LIN {X 0,Y 313.862,Z 653.442,A -85,B 0,C 180,E1 -16164.593,E2 -16164.593} C_VEL
LIN {X 0,Y 312.967,Z 666.014,A -85,B 0,C 180,E1 -16165.653,E2 -16165.653} C_VEL
LIN {X 0,Y 311.886,Z 679.603,A -85,B 0,C 180,E1 -16167.108,E2 -16167.108} C_VEL
LIN {X 0,Y 310.731,Z 691.302,A -85,B 0,C 180,E1 -16168.655,E2 -16168.655} C_VEL
LIN {X 0,Y 309.643,Z 702.145,A -85,B 0,C 180,E1 -16170.419,E2 -16170.419} C_VEL
LIN {X 0,Y 308.883,Z 708.95,A -85,B 0,C 180,E1 -16171.72,E2 -16171.72} C_VEL
LIN {X 0,Y 307.8,Z 712.897,A -85,B 0,C 180,E1 -16172.513,E2 -16172.513} C_VEL
LIN {X 0,Y 304.339,Z 719.014,A -85,B 0,C 180,E1 -16173.825,E2 -16173.825} C_VEL
LIN {X 0,Y 300.937,Z 724.622,A -85,B 0,C 180,E1 -16175.238,E2 -16175.238} C_VEL
LIN {X 0,Y 299.968,Z 727.754,A -85,B 0,C 180,E1 -16176.177,E2 -16176.177} C_VEL
LIN {X 0,Y 299.269,Z 734.632,A -85,B 0,C 180,E1 -16178.655,E2 -16178.655} C_VEL
LIN {X 0,Y 298.891,Z 739.258,A -85,B 0,C 180,E1 -16180.781,E2 -16180.781} C_VEL
LIN {X 0,Y 298.646,Z 742.834,A -85,B 0,C 180,E1 -16182.893,E2 -16182.893} C_VEL
LIN {X 0,Y 298.627,Z 745.46,A -85,B 0,C 180,E1 -16184.997,E2 -16184.997} C_VEL
LIN {X 0,Y 298.833,Z 747.584,A -85,B 0,C 180,E1 -16187.781,E2 -16187.781} C_VEL
LIN {X 0,Y 299.31,Z 748.208,A -85,B 0,C 180,E1 -16190.54,E2 -16190.54} C_VEL
LIN {X 0,Y 300.074,Z 747.31,A -85,B 0,C 180,E1 -16193.276,E2 -16193.276} C_VEL
LIN {X 0,Y 301.251,Z 744.941,A -85,B 0,C 180,E1 -16195.987,E2 -16195.987} C_VEL
LIN {X 0,Y 302.374,Z 742.07,A -85,B 0,C 180,E1 -16198.047,E2 -16198.047} C_VEL
LIN {X 0,Y 304.129,Z 737.027,A -85,B 0,C 180,E1 -16200.663,E2 -16200.663} C_VEL
LIN {X 0,Y 305.674,Z 732.008,A -85,B 0,C 180,E1 -16202.636,E2 -16202.636} C_VEL
LIN {X 0,Y 307.809,Z 724.674,A -85,B 0,C 180,E1 -16204.912,E2 -16204.912} C_VEL
LIN {X 0,Y 309.873,Z 716.852,A -85,B 0,C 180,E1 -16206.839,E2 -16206.839} C_VEL
LIN {X 0,Y 312.038,Z 707.448,A -85,B 0,C 180,E1 -16208.745,E2 -16208.745} C_VEL
LIN {X 0,Y 314.263,Z 696.794,A -85,B 0,C 180,E1 -16210.486,E2 -16210.486} C_VEL
LIN {X 0,Y 316.318,Z 685.009,A -85,B 0,C 180,E1 -16212.023,E2 -16212.023} C_VEL
LIN {X 0,Y 318.24,Z 671.492,A -85,B 0,C 180,E1 -16213.408,E2 -16213.408} C_VEL
LIN {X 0,Y 319.562,Z 658.715,A -85,B 0,C 180,E1 -16214.439,E2 -16214.439} C_VEL
LIN {X 0,Y 320.44,Z 645.691,A -85,B 0,C 180,E1 -16215.235,E2 -16215.235} C_VEL
LIN {X 0,Y 320.888,Z 631.299,A -85,B 0,C 180,E1 -16215.863,E2 -16215.863} C_VEL
LIN {X 0,Y 322.128,Z 601.129,A -85,B 0,C 180,E1 -16216.863,E2 -16216.863} C_VEL
LIN {X 0,Y 317.545,Z 592.238,A -85,B 0,C 180,E1 -16218.074,E2 -16218.074} C_VEL
LIN {X 0,Y 311.17,Z 581.718,A -85,B 0,C 180,E1 -16219.887,E2 -16219.887} C_VEL
LIN {X 0,Y 308.467,Z 577.764,A -85,B 0,C 180,E1 -16220.724,E2 -16220.724} C_VEL
LIN {X 0,Y 306.134,Z 574.422,A -85,B 0,C 180,E1 -16221.491,E2 -16221.491} C_VEL
LIN {X 0,Y 305.23,Z 573.248,A -85,B 0,C 180,E1 -16221.792,E2 -16221.792} C_VEL
LIN {X 0,Y 302.984,Z 570.401,A -85,B 0,C 180,E1 -16222.579,E2 -16222.579} C_VEL
LIN {X 0,Y 302.035,Z 568.615,A -85,B 0,C 180,E1 -16222.97,E2 -16222.97} C_VEL
LIN {X 0,Y 299.778,Z 566.635,A -85,B 0,C 180,E1 -16223.784,E2 -16223.784} C_VEL
LIN {X 0,Y 298.652,Z 564.26,A -85,B 0,C 180,E1 -16224.329,E2 -16224.329} C_VEL
LIN {X 0,Y 298.46,Z 563.308,A -85,B 0,C 180,E1 -16224.494,E2 -16224.494} C_VEL
LIN {X 0,Y 298.467,Z 563.298,A -85,B 0,C 180,E1 -16228.096,E2 -16228.096} C_VEL
LIN {X 0,Y 298.393,Z 563.303,A -85,B 0,C 180,E1 -16232.018,E2 -16232.018} C_VEL
LIN {X 0,Y 298.417,Z 563.307,A -85,B 0,C 180,E1 -16236.071,E2 -16236.071} C_VEL
LIN {X 0,Y 298.407,Z 563.307,A -85,B 0,C 180,E1 -16239.487,E2 -16239.487} C_VEL
LIN {X 0,Y 298.397,Z 563.316,A -85,B 0,C 180,E1 -16243.104,E2 -16243.104} C_VEL
LIN {X 0,Y 298.402,Z 563.315,A -85,B 0,C 180,E1 -16246.922,E2 -16246.922} C_VEL
LIN {X 0,Y 298.492,Z 563.489,A -85,B 0,C 180,E1 -16249.649,E2 -16249.649} C_VEL
LIN {X 0,Y 301.141,Z 576.792,A -85,B 0,C 180,E1 -16253.9,E2 -16253.9} C_VEL
LIN {X 0,Y 301.399,Z 577.984,A -85,B 0,C 180,E1 -16254.154,E2 -16254.154} C_VEL
LIN {X 0,Y 303.56,Z 584.867,A -85,B 0,C 180,E1 -16255.203,E2 -16255.203} C_VEL
LIN {X 0,Y 306.105,Z 590.438,A -85,B 0,C 180,E1 -16256.206,E2 -16256.206} C_VEL
LIN {X 0,Y 307.177,Z 596.338,A -85,B 0,C 180,E1 -16256.808,E2 -16256.808} C_VEL
LIN {X 0,Y 309.228,Z 608.134,A -85,B 0,C 180,E1 -16257.935,E2 -16257.935} C_VEL
LIN {X 0,Y 311.234,Z 620.326,A -85,B 0,C 180,E1 -16258.994,E2 -16258.994} C_VEL
LIN {X 0,Y 313.643,Z 638.097,A -85,B 0,C 180,E1 -16260.348,E2 -16260.348} C_VEL
LIN {X 0,Y 315.127,Z 652.445,A -85,B 0,C 180,E1 -16261.291,E2 -16261.291} C_VEL
LIN {X 0,Y 316.933,Z 687.14,A -85,B 0,C 180,E1 -16263.131,E2 -16263.131} C_VEL
LIN {X 0,Y 314.907,Z 716.371,A -85,B 0,C 180,E1 -16264.158,E2 -16264.158} C_VEL
LIN {X 0,Y 313.288,Z 730.542,A -85,B 0,C 180,E1 -16264.861,E2 -16264.861} C_VEL
LIN {X 0,Y 311.103,Z 744.781,A -85,B 0,C 180,E1 -16265.83,E2 -16265.83} C_VEL
LIN {X 0,Y 308.923,Z 756.894,A -85,B 0,C 180,E1 -16266.895,E2 -16266.895} C_VEL
LIN {X 0,Y 306.369,Z 769.537,A -85,B 0,C 180,E1 -16268.291,E2 -16268.291} C_VEL
LIN {X 0,Y 303.751,Z 782.108,A -85,B 0,C 180,E1 -16270.046,E2 -16270.046} C_VEL
LIN {X 0,Y 301.798,Z 791.503,A -85,B 0,C 180,E1 -16271.678,E2 -16271.678} C_VEL
LIN {X 0,Y 300.046,Z 800.913,A -85,B 0,C 180,E1 -16273.676,E2 -16273.676} C_VEL
LIN {X 0,Y 298.759,Z 808.708,A -85,B 0,C 180,E1 -16275.701,E2 -16275.701} C_VEL
LIN {X 0,Y 297.902,Z 815.115,A -85,B 0,C 180,E1 -16277.742,E2 -16277.742} C_VEL
LIN {X 0,Y 297.452,Z 820.325,A -85,B 0,C 180,E1 -16279.794,E2 -16279.794} C_VEL
LIN {X 0,Y 297.448,Z 824.422,A -85,B 0,C 180,E1 -16281.851,E2 -16281.851} C_VEL
LIN {X 0,Y 297.554,Z 826.59,A -85,B 0,C 180,E1 -16283.219,E2 -16283.219} C_VEL
LIN {X 0,Y 297.84,Z 828.297,A -85,B 0,C 180,E1 -16284.585,E2 -16284.585} C_VEL
LIN {X 0,Y 298.066,Z 829.525,A -85,B 0,C 180,E1 -16285.945,E2 -16285.945} C_VEL
LIN {X 0,Y 298.48,Z 831.378,A -85,B 0,C 180,E1 -16288.652,E2 -16288.652} C_VEL
LIN {X 0,Y 298.642,Z 832.113,A -85,B 0,C 180,E1 -16290.001,E2 -16290.001} C_VEL
LIN {X 0,Y 298.292,Z 832.305,A -85,B 0,C 180,E1 -16291.351,E2 -16291.351} C_VEL
LIN {X 0,Y 298.009,Z 832.056,A -85,B 0,C 180,E1 -16292.704,E2 -16292.704} C_VEL
LIN {X 0,Y 297.877,Z 831.381,A -85,B 0,C 180,E1 -16294.06,E2 -16294.06} C_VEL
LIN {X 0,Y 297.6,Z 830.213,A -85,B 0,C 180,E1 -16295.421,E2 -16295.421} C_VEL
LIN {X 0,Y 297.401,Z 828.284,A -85,B 0,C 180,E1 -16297.009,E2 -16297.009} C_VEL
LIN {X 0,Y 297.267,Z 824.044,A -85,B 0,C 180,E1 -16299.527,E2 -16299.527} C_VEL
LIN {X 0,Y 297.59,Z 819.438,A -85,B 0,C 180,E1 -16301.581,E2 -16301.581} C_VEL
LIN {X 0,Y 298.452,Z 812.667,A -85,B 0,C 180,E1 -16303.968,E2 -16303.968} C_VEL
LIN {X 0,Y 299.924,Z 804.235,A -85,B 0,C 180,E1 -16306.332,E2 -16306.332} C_VEL
LIN {X 0,Y 301.817,Z 795.451,A -85,B 0,C 180,E1 -16308.323,E2 -16308.323} C_VEL
LIN {X 0,Y 304.397,Z 784.963,A -85,B 0,C 180,E1 -16310.263,E2 -16310.263} C_VEL
LIN {X 0,Y 307.345,Z 772.409,A -85,B 0,C 180,E1 -16312.167,E2 -16312.167} C_VEL
LIN {X 0,Y 310.337,Z 759.719,A -85,B 0,C 180,E1 -16313.702,E2 -16313.702} C_VEL
LIN {X 0,Y 313.806,Z 744.255,A -85,B 0,C 180,E1 -16315.185,E2 -16315.185} C_VEL
LIN {X 0,Y 317.017,Z 727.607,A -85,B 0,C 180,E1 -16316.409,E2 -16316.409} C_VEL
LIN {X 0,Y 319.563,Z 711.784,A -85,B 0,C 180,E1 -16317.285,E2 -16317.285} C_VEL
LIN {X 0,Y 321.41,Z 694.915,A -85,B 0,C 180,E1 -16318.002,E2 -16318.002} C_VEL
LIN {X 0,Y 322.095,Z 686.631,A -85,B 0,C 180,E1 -16318.306,E2 -16318.306} C_VEL
LIN {X 0,Y 322.687,Z 658.06,A -85,B 0,C 180,E1 -16319.736,E2 -16319.736} C_VEL
LIN {X 0,Y 322.259,Z 641.073,A -85,B 0,C 180,E1 -16320.812,E2 -16320.812} C_VEL
LIN {X 0,Y 321.121,Z 625.091,A -85,B 0,C 180,E1 -16322.077,E2 -16322.077} C_VEL
LIN {X 0,Y 319.501,Z 609.013,A -85,B 0,C 180,E1 -16323.616,E2 -16323.616} C_VEL
LIN {X 0,Y 317.914,Z 596.006,A -85,B 0,C 180,E1 -16325.12,E2 -16325.12} C_VEL
LIN {X 0,Y 317.288,Z 592.328,A -85,B 0,C 180,E1 -16325.646,E2 -16325.646} C_VEL
LIN {X 0,Y 315.159,Z 584.693,A -85,B 0,C 180,E1 -16327.186,E2 -16327.186} C_VEL
LIN {X 0,Y 313.05,Z 581.45,A -85,B 0,C 180,E1 -16328.542,E2 -16328.542} C_VEL
LIN {X 0,Y 312.505,Z 580.505,A -85,B 0,C 180,E1 -16328.947,E2 -16328.947} C_VEL
LIN {X 0,Y 310.14,Z 578.285,A -85,B 0,C 180,E1 -16330.8,E2 -16330.8} C_VEL
LIN {X 0,Y 309.024,Z 575.541,A -85,B 0,C 180,E1 -16332.369,E2 -16332.369} C_VEL
LIN {X 0,Y 308.515,Z 575.136,A -85,B 0,C 180,E1 -16333.111,E2 -16333.111} C_VEL
LIN {X 0,Y 307.708,Z 574.825,A -85,B 0,C 180,E1 -16335.076,E2 -16335.076} C_VEL
LIN {X 0,Y 308.083,Z 574.969,A -85,B 0,C 180,E1 -16337.823,E2 -16337.823} C_VEL
LIN {X 0,Y 309.094,Z 575.419,A -85,B 0,C 180,E1 -16339.393,E2 -16339.393} C_VEL
LIN {X 0,Y 310.311,Z 578.396,A -85,B 0,C 180,E1 -16341.026,E2 -16341.026} C_VEL
LIN {X 0,Y 313.048,Z 580.971,A -85,B 0,C 180,E1 -16343.017,E2 -16343.017} C_VEL
LIN {X 0,Y 315.136,Z 584.426,A -85,B 0,C 180,E1 -16344.323,E2 -16344.323} C_VEL
LIN {X 0,Y 316.493,Z 585.995,A -85,B 0,C 180,E1 -16345.026,E2 -16345.026} C_VEL
LIN {X 0,Y 318.779,Z 589.401,A -85,B 0,C 180,E1 -16346.114,E2 -16346.114} C_VEL
LIN {X 0,Y 322.345,Z 594.975,A -85,B 0,C 180,E1 -16347.583,E2 -16347.583} C_VEL
LIN {X 0,Y 326.335,Z 601.805,A -85,B 0,C 180,E1 -16349.012,E2 -16349.012} C_VEL
LIN {X 0,Y 328.926,Z 606.977,A -85,B 0,C 180,E1 -16349.872,E2 -16349.872} C_VEL
LIN {X 0,Y 327.816,Z 633.197,A -85,B 0,C 180,E1 -16350.905,E2 -16350.905} C_VEL
LIN {X 0,Y 326.745,Z 649.064,A -85,B 0,C 180,E1 -16351.798,E2 -16351.798} C_VEL
LIN {X 0,Y 325.289,Z 662.738,A -85,B 0,C 180,E1 -16352.819,E2 -16352.819} C_VEL
LIN {X 0,Y 323.603,Z 673.85,A -85,B 0,C 180,E1 -16353.843,E2 -16353.843} C_VEL
LIN {X 0,Y 321.425,Z 686.452,A -85,B 0,C 180,E1 -16355.28,E2 -16355.28} C_VEL
LIN {X 0,Y 319.03,Z 697.533,A -85,B 0,C 180,E1 -16356.81,E2 -16356.81} C_VEL
LIN {X 0,Y 316.512,Z 707.592,A -85,B 0,C 180,E1 -16358.507,E2 -16358.507} C_VEL
LIN {X 0,Y 313.936,Z 716.841,A -85,B 0,C 180,E1 -16360.378,E2 -16360.378} C_VEL
LIN {X 0,Y 311.167,Z 725.674,A -85,B 0,C 180,E1 -16362.586,E2 -16362.586} C_VEL
LIN {X 0,Y 308.638,Z 732.86,A -85,B 0,C 180,E1 -16364.819,E2 -16364.819} C_VEL
LIN {X 0,Y 306.169,Z 739.408,A -85,B 0,C 180,E1 -16367.404,E2 -16367.404} C_VEL
LIN {X 0,Y 303.97,Z 744.389,A -85,B 0,C 180,E1 -16370.014,E2 -16370.014} C_VEL
LIN {X 0,Y 302.806,Z 747.144,A -85,B 0,C 180,E1 -16371.995,E2 -16371.995} C_VEL
LIN {X 0,Y 301.357,Z 749.7,A -85,B 0,C 180,E1 -16374.647,E2 -16374.647} C_VEL
LIN {X 0,Y 300.28,Z 750.965,A -85,B 0,C 180,E1 -16377.316,E2 -16377.316} C_VEL
LIN {X 0,Y 299.539,Z 750.972,A -85,B 0,C 180,E1 -16379.999,E2 -16379.999} C_VEL
LIN {X 0,Y 298.994,Z 749.742,A -85,B 0,C 180,E1 -16382.694,E2 -16382.694} C_VEL
LIN {X 0,Y 298.714,Z 747.243,A -85,B 0,C 180,E1 -16385.399,E2 -16385.399} C_VEL
LIN {X 0,Y 298.943,Z 744.448,A -85,B 0,C 180,E1 -16387.429,E2 -16387.429} C_VEL
LIN {X 0,Y 299.139,Z 739.571,A -85,B 0,C 180,E1 -16390.148,E2 -16390.148} C_VEL
LIN {X 0,Y 299.603,Z 733.169,A -85,B 0,C 180,E1 -16392.876,E2 -16392.876} C_VEL
LIN {X 0,Y 300.328,Z 726.129,A -85,B 0,C 180,E1 -16395.263,E2 -16395.263} C_VEL
LIN {X 0,Y 301.208,Z 717.545,A -85,B 0,C 180,E1 -16397.657,E2 -16397.657} C_VEL
LIN {X 0,Y 302.148,Z 708.694,A -85,B 0,C 180,E1 -16399.71,E2 -16399.71} C_VEL
LIN {X 0,Y 303.365,Z 698.188,A -85,B 0,C 180,E1 -16401.756,E2 -16401.756} C_VEL
LIN {X 0,Y 304.585,Z 686.663,A -85,B 0,C 180,E1 -16403.634,E2 -16403.634} C_VEL
LIN {X 0,Y 305.896,Z 674.092,A -85,B 0,C 180,E1 -16405.334,E2 -16405.334} C_VEL
LIN {X 0,Y 307.004,Z 661.206,A -85,B 0,C 180,E1 -16406.772,E2 -16406.772} C_VEL
LIN {X 0,Y 308.111,Z 646.816,A -85,B 0,C 180,E1 -16408.063,E2 -16408.063} C_VEL
LIN {X 0,Y 308.927,Z 632.193,A -85,B 0,C 180,E1 -16409.095,E2 -16409.095} C_VEL
LIN {X 0,Y 309.637,Z 616.184,A -85,B 0,C 180,E1 -16409.928,E2 -16409.928} C_VEL
LIN {X 0,Y 309.824,Z 594.608,A -85,B 0,C 180,E1 -16410.698,E2 -16410.698} C_VEL
LIN {X 0,Y 298.475,Z 563.631,A -85,B 0,C 180,E1 -16412.431,E2 -16412.431} C_VEL
LIN {X 0,Y 298.435,Z 563.31,A -85,B 0,C 180,E1 -16412.475,E2 -16412.475} C_VEL
LIN {X 0,Y 298.42,Z 563.314,A -85,B 0,C 180,E1 -16416.069,E2 -16416.069} C_VEL
LIN {X 0,Y 298.409,Z 563.311,A -85,B 0,C 180,E1 -16419.485,E2 -16419.485} C_VEL
LIN {X 0,Y 298.399,Z 563.312,A -85,B 0,C 180,E1 -16423.102,E2 -16423.102} C_VEL
LIN {X 0,Y 298.403,Z 563.312,A -85,B 0,C 180,E1 -16426.92,E2 -16426.92} C_VEL
LIN {X 0,Y 298.415,Z 563.311,A -85,B 0,C 180,E1 -16431.003,E2 -16431.003} C_VEL
LIN {X 0,Y 298.432,Z 563.309,A -85,B 0,C 180,E1 -16433.931,E2 -16433.931} C_VEL
LIN {X 0,Y 298.393,Z 563.313,A -85,B 0,C 180,E1 -16437.983,E2 -16437.983} C_VEL
LIN {X 0,Y 298.456,Z 563.305,A -85,B 0,C 180,E1 -16441.903,E2 -16441.903} C_VEL
LIN {X 0,Y 298.482,Z 563.304,A -85,B 0,C 180,E1 -16444.923,E2 -16444.923} C_VEL
LIN {X 0,Y 298.449,Z 563.307,A -85,B 0,C 180,E1 -16449.314,E2 -16449.314} C_VEL
LIN {X 0,Y 298.537,Z 563.295,A -85,B 0,C 180,E1 -16452.179,E2 -16452.179} C_VEL
LIN {X 0,Y 298.592,Z 563.292,A -85,B 0,C 180,E1 -16454.994,E2 -16454.994} C_VEL
LIN {X 0,Y 298.592,Z 563.292,A -85,B 0,C 180,E1 -16459.146,E2 -16459.146} C_VEL
LIN {X 0,Y 298.756,Z 563.267,A -85,B 0,C 180,E1 -16461.885,E2 -16461.885} C_VEL
LIN {X 0,Y 298.659,Z 563.28,A -85,B 0,C 180,E1 -16464.598,E2 -16464.598} C_VEL
LIN {X 0,Y 298.922,Z 563.248,A -85,B 0,C 180,E1 -16468.652,E2 -16468.652} C_VEL
LIN {X 0,Y 298.922,Z 563.25,A -85,B 0,C 180,E1 -16471.346,E2 -16471.346} C_VEL
LIN {X 0,Y 298.794,Z 563.264,A -85,B 0,C 180,E1 -16476.753,E2 -16476.753} C_VEL
LIN {X 0,Y 298.678,Z 563.281,A -85,B 0,C 180,E1 -16479.48,E2 -16479.48} C_VEL
LIN {X 0,Y 298.551,Z 563.296,A -85,B 0,C 180,E1 -16483.615,E2 -16483.615} C_VEL
LIN {X 0,Y 298.545,Z 563.294,A -85,B 0,C 180,E1 -16486.408,E2 -16486.408} C_VEL
LIN {X 0,Y 298.508,Z 563.302,A -85,B 0,C 180,E1 -16489.654,E2 -16489.654} C_VEL
LIN {X 0,Y 298.453,Z 563.311,A -85,B 0,C 180,E1 -16493.597,E2 -16493.597} C_VEL
LIN {X 0,Y 298.485,Z 563.301,A -85,B 0,C 180,E1 -16496.574,E2 -16496.574} C_VEL
LIN {X 0,Y 298.417,Z 563.314,A -85,B 0,C 180,E1 -16499.64,E2 -16499.64} C_VEL
LIN {X 0,Y 298.393,Z 563.313,A -85,B 0,C 180,E1 -16502.799,E2 -16502.799} C_VEL
LIN {X 0,Y 298.465,Z 563.304,A -85,B 0,C 180,E1 -16506.814,E2 -16506.814} C_VEL
LIN {X 0,Y 298.414,Z 563.31,A -85,B 0,C 180,E1 -16511.095,E2 -16511.095} C_VEL
LIN {X 0,Y 298.474,Z 563.303,A -85,B 0,C 180,E1 -16515.059,E2 -16515.059} C_VEL
LIN {X 0,Y 298.451,Z 563.306,A -85,B 0,C 180,E1 -16518.897,E2 -16518.897} C_VEL
LIN {X 0,Y 298.484,Z 563.337,A -85,B 0,C 180,E1 -16520.126,E2 -16520.126} C_VEL
LIN {X 0,Y 308.877,Z 591.597,A -85,B 0,C 180,E1 -16521.648,E2 -16521.648} C_VEL
LIN {X 0,Y 308.12,Z 626.263,A -85,B 0,C 180,E1 -16522.716,E2 -16522.716} C_VEL
LIN {X 0,Y 307.657,Z 641.211,A -85,B 0,C 180,E1 -16523.429,E2 -16523.429} C_VEL
LIN {X 0,Y 306.945,Z 655.249,A -85,B 0,C 180,E1 -16524.379,E2 -16524.379} C_VEL
LIN {X 0,Y 305.997,Z 667.921,A -85,B 0,C 180,E1 -16525.489,E2 -16525.489} C_VEL
LIN {X 0,Y 304.974,Z 680.056,A -85,B 0,C 180,E1 -16526.818,E2 -16526.818} C_VEL
LIN {X 0,Y 303.838,Z 691.52,A -85,B 0,C 180,E1 -16528.353,E2 -16528.353} C_VEL
LIN {X 0,Y 302.768,Z 702.038,A -85,B 0,C 180,E1 -16530.062,E2 -16530.062} C_VEL
LIN {X 0,Y 301.753,Z 711.228,A -85,B 0,C 180,E1 -16531.86,E2 -16531.86} C_VEL
LIN {X 0,Y 300.726,Z 720.293,A -85,B 0,C 180,E1 -16534.012,E2 -16534.012} C_VEL
LIN {X 0,Y 299.968,Z 727.754,A -85,B 0,C 180,E1 -16536.177,E2 -16536.177} C_VEL
LIN {X 0,Y 299.025,Z 730.738,A -85,B 0,C 180,E1 -16537.137,E2 -16537.137} C_VEL
LIN {X 0,Y 295.772,Z 735.312,A -85,B 0,C 180,E1 -16538.713,E2 -16538.713} C_VEL
LIN {X 0,Y 292.568,Z 739.32,A -85,B 0,C 180,E1 -16540.373,E2 -16540.373} C_VEL
LIN {X 0,Y 291.73,Z 741.402,A -85,B 0,C 180,E1 -16541.449,E2 -16541.449} C_VEL
LIN {X 0,Y 291.601,Z 744.163,A -85,B 0,C 180,E1 -16543.19,E2 -16543.19} C_VEL
LIN {X 0,Y 291.589,Z 745.998,A -85,B 0,C 180,E1 -16544.626,E2 -16544.626} C_VEL
LIN {X 0,Y 291.773,Z 748.412,A -85,B 0,C 180,E1 -16547.48,E2 -16547.48} C_VEL
LIN {X 0,Y 292.276,Z 749.327,A -85,B 0,C 180,E1 -16550.352,E2 -16550.352} C_VEL
LIN {X 0,Y 293.036,Z 748.778,A -85,B 0,C 180,E1 -16553.113,E2 -16553.113} C_VEL
LIN {X 0,Y 294.235,Z 746.691,A -85,B 0,C 180,E1 -16555.891,E2 -16555.891} C_VEL
LIN {X 0,Y 295.782,Z 743.113,A -85,B 0,C 180,E1 -16558.639,E2 -16558.639} C_VEL
LIN {X 0,Y 297.213,Z 739.357,A -85,B 0,C 180,E1 -16560.678,E2 -16560.678} C_VEL
LIN {X 0,Y 298.841,Z 734.612,A -85,B 0,C 180,E1 -16562.697,E2 -16562.697} C_VEL
LIN {X 0,Y 301.002,Z 727.665,A -85,B 0,C 180,E1 -16565.024,E2 -16565.024} C_VEL
LIN {X 0,Y 303.176,Z 720.305,A -85,B 0,C 180,E1 -16566.991,E2 -16566.991} C_VEL
LIN {X 0,Y 305.499,Z 711.385,A -85,B 0,C 180,E1 -16568.934,E2 -16568.934} C_VEL
LIN {X 0,Y 307.74,Z 701.378,A -85,B 0,C 180,E1 -16570.694,E2 -16570.694} C_VEL
LIN {X 0,Y 310.152,Z 689.323,A -85,B 0,C 180,E1 -16572.396,E2 -16572.396} C_VEL
LIN {X 0,Y 312.041,Z 677.987,A -85,B 0,C 180,E1 -16573.68,E2 -16573.68} C_VEL
LIN {X 0,Y 313.529,Z 666.001,A -85,B 0,C 180,E1 -16574.773,E2 -16574.773} C_VEL
LIN {X 0,Y 314.715,Z 652.143,A -85,B 0,C 180,E1 -16575.746,E2 -16575.746} C_VEL
LIN {X 0,Y 315.472,Z 637.83,A -85,B 0,C 180,E1 -16576.472,E2 -16576.472} C_VEL
LIN {X 0,Y 316.684,Z 609.568,A -85,B 0,C 180,E1 -16577.467,E2 -16577.467} C_VEL
LIN {X 0,Y 316.905,Z 603.833,A -85,B 0,C 180,E1 -16577.679,E2 -16577.679} C_VEL
LIN {X 0,Y 312.007,Z 594.49,A -85,B 0,C 180,E1 -16579.072,E2 -16579.072} C_VEL
LIN {X 0,Y 307.005,Z 586.324,A -85,B 0,C 180,E1 -16580.606,E2 -16580.606} C_VEL
LIN {X 0,Y 304.838,Z 583.128,A -85,B 0,C 180,E1 -16581.316,E2 -16581.316} C_VEL
LIN {X 0,Y 302.322,Z 579.392,A -85,B 0,C 180,E1 -16582.2,E2 -16582.2} C_VEL
LIN {X 0,Y 299.816,Z 576.022,A -85,B 0,C 180,E1 -16583.137,E2 -16583.137} C_VEL
LIN {X 0,Y 298.89,Z 574.638,A -85,B 0,C 180,E1 -16583.507,E2 -16583.507} C_VEL
LIN {X 0,Y 296.511,Z 571.918,A -85,B 0,C 180,E1 -16584.483,E2 -16584.483} C_VEL
LIN {X 0,Y 295.5,Z 569.723,A -85,B 0,C 180,E1 -16584.997,E2 -16584.997} C_VEL
LIN {X 0,Y 293.007,Z 567.834,A -85,B 0,C 180,E1 -16586.102,E2 -16586.102} C_VEL
LIN {X 0,Y 291.615,Z 565.117,A -85,B 0,C 180,E1 -16586.913,E2 -16586.913} C_VEL
LIN {X 0,Y 291.415,Z 564.179,A -85,B 0,C 180,E1 -16587.103,E2 -16587.103} C_VEL
LIN {X 0,Y 291.335,Z 564.184,A -85,B 0,C 180,E1 -16590.438,E2 -16590.438} C_VEL
LIN {X 0,Y 291.343,Z 564.186,A -85,B 0,C 180,E1 -16593.699,E2 -16593.699} C_VEL
LIN {X 0,Y 291.379,Z 564.18,A -85,B 0,C 180,E1 -16597.256,E2 -16597.256} C_VEL
LIN {X 0,Y 291.333,Z 564.195,A -85,B 0,C 180,E1 -16600.643,E2 -16600.643} C_VEL
LIN {X 0,Y 291.313,Z 564.195,A -85,B 0,C 180,E1 -16604.398,E2 -16604.398} C_VEL
LIN {X 0,Y 291.348,Z 564.182,A -85,B 0,C 180,E1 -16608.4,E2 -16608.4} C_VEL
LIN {X 0,Y 291.455,Z 564.348,A -85,B 0,C 180,E1 -16609.48,E2 -16609.48} C_VEL
LIN {X 0,Y 294.347,Z 574.648,A -85,B 0,C 180,E1 -16611.605,E2 -16611.605} C_VEL
LIN {X 0,Y 297.819,Z 582.824,A -85,B 0,C 180,E1 -16613.416,E2 -16613.416} C_VEL
LIN {X 0,Y 299.953,Z 589.964,A -85,B 0,C 180,E1 -16614.557,E2 -16614.557} C_VEL
LIN {X 0,Y 301.952,Z 594.666,A -85,B 0,C 180,E1 -16615.41,E2 -16615.41} C_VEL
LIN {X 0,Y 303.256,Z 602.424,A -85,B 0,C 180,E1 -16616.229,E2 -16616.229} C_VEL
LIN {X 0,Y 305.319,Z 615.028,A -85,B 0,C 180,E1 -16617.456,E2 -16617.456} C_VEL
LIN {X 0,Y 307.777,Z 632.99,A -85,B 0,C 180,E1 -16618.973,E2 -16618.973} C_VEL
LIN {X 0,Y 309.841,Z 652.667,A -85,B 0,C 180,E1 -16620.387,E2 -16620.387} C_VEL
LIN {X 0,Y 311.4,Z 688.271,A -85,B 0,C 180,E1 -16622.345,E2 -16622.345} C_VEL
LIN {X 0,Y 309.461,Z 714.825,A -85,B 0,C 180,E1 -16623.306,E2 -16623.306} C_VEL
LIN {X 0,Y 307.73,Z 728.782,A -85,B 0,C 180,E1 -16624.011,E2 -16624.011} C_VEL
LIN {X 0,Y 305.408,Z 742.927,A -85,B 0,C 180,E1 -16624.987,E2 -16624.987} C_VEL
LIN {X 0,Y 302.77,Z 756.697,A -85,B 0,C 180,E1 -16626.215,E2 -16626.215} C_VEL
LIN {X 0,Y 300.125,Z 769.04,A -85,B 0,C 180,E1 -16627.635,E2 -16627.635} C_VEL
LIN {X 0,Y 297.533,Z 780.339,A -85,B 0,C 180,E1 -16629.25,E2 -16629.25} C_VEL
LIN {X 0,Y 295.06,Z 791.503,A -85,B 0,C 180,E1 -16631.244,E2 -16631.244} C_VEL
LIN {X 0,Y 293.193,Z 800.689,A -85,B 0,C 180,E1 -16633.284,E2 -16633.284} C_VEL
LIN {X 0,Y 291.851,Z 808.294,A -85,B 0,C 180,E1 -16635.355,E2 -16635.355} C_VEL
LIN {X 0,Y 290.909,Z 814.567,A -85,B 0,C 180,E1 -16637.443,E2 -16637.443} C_VEL
LIN {X 0,Y 290.408,Z 819.631,A -85,B 0,C 180,E1 -16639.544,E2 -16639.544} C_VEL
LIN {X 0,Y 290.355,Z 823.613,A -85,B 0,C 180,E1 -16641.65,E2 -16641.65} C_VEL
LIN {X 0,Y 290.461,Z 825.705,A -85,B 0,C 180,E1 -16643.052,E2 -16643.052} C_VEL
LIN {X 0,Y 290.731,Z 827.33,A -85,B 0,C 180,E1 -16644.452,E2 -16644.452} C_VEL
LIN {X 0,Y 291.004,Z 828.522,A -85,B 0,C 180,E1 -16645.846,E2 -16645.846} C_VEL
LIN {X 0,Y 291.48,Z 830.06,A -85,B 0,C 180,E1 -16648.619,E2 -16648.619} C_VEL
LIN {X 0,Y 291.653,Z 830.896,A -85,B 0,C 180,E1 -16650.001,E2 -16650.001} C_VEL
LIN {X 0,Y 291.271,Z 831.136,A -85,B 0,C 180,E1 -16651.383,E2 -16651.383} C_VEL
LIN {X 0,Y 290.975,Z 830.944,A -85,B 0,C 180,E1 -16652.77,E2 -16652.77} C_VEL
LIN {X 0,Y 290.819,Z 830.321,A -85,B 0,C 180,E1 -16654.158,E2 -16654.158} C_VEL
LIN {X 0,Y 290.513,Z 829.236,A -85,B 0,C 180,E1 -16655.554,E2 -16655.554} C_VEL
LIN {X 0,Y 290.329,Z 827.629,A -85,B 0,C 180,E1 -16657.023,E2 -16657.023} C_VEL
LIN {X 0,Y 290.218,Z 823.321,A -85,B 0,C 180,E1 -16659.76,E2 -16659.76} C_VEL
LIN {X 0,Y 290.586,Z 818.876,A -85,B 0,C 180,E1 -16661.864,E2 -16661.864} C_VEL
LIN {X 0,Y 291.506,Z 812.298,A -85,B 0,C 180,E1 -16664.308,E2 -16664.308} C_VEL
LIN {X 0,Y 292.591,Z 806.094,A -85,B 0,C 180,E1 -16666.194,E2 -16666.194} C_VEL
LIN {X 0,Y 294.717,Z 797.151,A -85,B 0,C 180,E1 -16668.42,E2 -16668.42} C_VEL
LIN {X 0,Y 297.248,Z 787.352,A -85,B 0,C 180,E1 -16670.411,E2 -16670.411} C_VEL
LIN {X 0,Y 300.345,Z 775.655,A -85,B 0,C 180,E1 -16672.35,E2 -16672.35} C_VEL
LIN {X 0,Y 303.596,Z 762.711,A -85,B 0,C 180,E1 -16674.08,E2 -16674.08} C_VEL
LIN {X 0,Y 307.15,Z 748.469,A -85,B 0,C 180,E1 -16675.588,E2 -16675.588} C_VEL
LIN {X 0,Y 310.243,Z 734.506,A -85,B 0,C 180,E1 -16676.759,E2 -16676.759} C_VEL
LIN {X 0,Y 313.336,Z 718.302,A -85,B 0,C 180,E1 -16677.829,E2 -16677.829} C_VEL
LIN {X 0,Y 315.983,Z 700.422,A -85,B 0,C 180,E1 -16678.695,E2 -16678.695} C_VEL
LIN {X 0,Y 317.18,Z 687,A -85,B 0,C 180,E1 -16679.244,E2 -16679.244} C_VEL
LIN {X 0,Y 318.04,Z 659.922,A -85,B 0,C 180,E1 -16680.634,E2 -16680.634} C_VEL
LIN {X 0,Y 317.869,Z 643.573,A -85,B 0,C 180,E1 -16681.7,E2 -16681.7} C_VEL
LIN {X 0,Y 316.969,Z 627.094,A -85,B 0,C 180,E1 -16683.05,E2 -16683.05} C_VEL
LIN {X 0,Y 315.629,Z 611.372,A -85,B 0,C 180,E1 -16684.634,E2 -16684.634} C_VEL
LIN {X 0,Y 314.469,Z 599.595,A -85,B 0,C 180,E1 -16686.045,E2 -16686.045} C_VEL
LIN {X 0,Y 314.02,Z 596.802,A -85,B 0,C 180,E1 -16686.481,E2 -16686.481} C_VEL
LIN {X 0,Y 312.52,Z 590.678,A -85,B 0,C 180,E1 -16687.752,E2 -16687.752} C_VEL
LIN {X 0,Y 310.403,Z 587.141,A -85,B 0,C 180,E1 -16689.291,E2 -16689.291} C_VEL
LIN {X 0,Y 307.989,Z 584.471,A -85,B 0,C 180,E1 -16691.434,E2 -16691.434} C_VEL
LIN {X 0,Y 307.307,Z 582.286,A -85,B 0,C 180,E1 -16692.656,E2 -16692.656} C_VEL
LIN {X 0,Y 306.175,Z 581.742,A -85,B 0,C 180,E1 -16695.365,E2 -16695.365} C_VEL
LIN {X 0,Y 306.599,Z 581.91,A -85,B 0,C 180,E1 -16697.794,E2 -16697.794} C_VEL
LIN {X 0,Y 307.42,Z 582.331,A -85,B 0,C 180,E1 -16699.161,E2 -16699.161} C_VEL
LIN {X 0,Y 308.735,Z 585.433,A -85,B 0,C 180,E1 -16700.96,E2 -16700.96} C_VEL
LIN {X 0,Y 311.063,Z 587.734,A -85,B 0,C 180,E1 -16702.705,E2 -16702.705} C_VEL
LIN {X 0,Y 313.197,Z 591.182,A -85,B 0,C 180,E1 -16704.102,E2 -16704.102} C_VEL
LIN {X 0,Y 314.223,Z 592.598,A -85,B 0,C 180,E1 -16704.683,E2 -16704.683} C_VEL
LIN {X 0,Y 317.08,Z 597.081,A -85,B 0,C 180,E1 -16706.089,E2 -16706.089} C_VEL
LIN {X 0,Y 319.789,Z 601.447,A -85,B 0,C 180,E1 -16707.232,E2 -16707.232} C_VEL
LIN {X 0,Y 323.705,Z 608.519,A -85,B 0,C 180,E1 -16708.713,E2 -16708.713} C_VEL
LIN {X 0,Y 324.444,Z 610.205,A -85,B 0,C 180,E1 -16708.991,E2 -16708.991} C_VEL
LIN {X 0,Y 323.085,Z 636.825,A -85,B 0,C 180,E1 -16710.097,E2 -16710.097} C_VEL
LIN {X 0,Y 321.923,Z 651.711,A -85,B 0,C 180,E1 -16710.982,E2 -16710.982} C_VEL
LIN {X 0,Y 320.384,Z 664.26,A -85,B 0,C 180,E1 -16711.95,E2 -16711.95} C_VEL
LIN {X 0,Y 318.451,Z 676.474,A -85,B 0,C 180,E1 -16713.1,E2 -16713.1} C_VEL
LIN {X 0,Y 316.41,Z 687.118,A -85,B 0,C 180,E1 -16714.333,E2 -16714.333} C_VEL
LIN {X 0,Y 313.841,Z 698.19,A -85,B 0,C 180,E1 -16715.877,E2 -16715.877} C_VEL
LIN {X 0,Y 311.422,Z 707.553,A -85,B 0,C 180,E1 -16717.44,E2 -16717.44} C_VEL
LIN {X 0,Y 308.909,Z 716.137,A -85,B 0,C 180,E1 -16719.154,E2 -16719.154} C_VEL
LIN {X 0,Y 306.019,Z 724.812,A -85,B 0,C 180,E1 -16721.244,E2 -16721.244} C_VEL
LIN {X 0,Y 303.659,Z 731.437,A -85,B 0,C 180,E1 -16723.183,E2 -16723.183} C_VEL
LIN {X 0,Y 301.488,Z 736.981,A -85,B 0,C 180,E1 -16725.142,E2 -16725.142} C_VEL
LIN {X 0,Y 298.924,Z 742.833,A -85,B 0,C 180,E1 -16727.783,E2 -16727.783} C_VEL
LIN {X 0,Y 296.758,Z 747.228,A -85,B 0,C 180,E1 -16730.457,E2 -16730.457} C_VEL
LIN {X 0,Y 295.182,Z 750.175,A -85,B 0,C 180,E1 -16733.162,E2 -16733.162} C_VEL
LIN {X 0,Y 293.812,Z 751.875,A -85,B 0,C 180,E1 -16735.884,E2 -16735.884} C_VEL
LIN {X 0,Y 292.881,Z 752.324,A -85,B 0,C 180,E1 -16738.624,E2 -16738.624} C_VEL
LIN {X 0,Y 292.24,Z 751.514,A -85,B 0,C 180,E1 -16741.377,E2 -16741.377} C_VEL
LIN {X 0,Y 291.821,Z 749.456,A -85,B 0,C 180,E1 -16744.143,E2 -16744.143} C_VEL
LIN {X 0,Y 291.891,Z 746.085,A -85,B 0,C 180,E1 -16746.914,E2 -16746.914} C_VEL
LIN {X 0,Y 292.043,Z 741.345,A -85,B 0,C 180,E1 -16749.697,E2 -16749.697} C_VEL
LIN {X 0,Y 292.465,Z 735.085,A -85,B 0,C 180,E1 -16752.49,E2 -16752.49} C_VEL
LIN {X 0,Y 293.12,Z 728.199,A -85,B 0,C 180,E1 -16754.936,E2 -16754.936} C_VEL
LIN {X 0,Y 293.984,Z 720.048,A -85,B 0,C 180,E1 -16757.315,E2 -16757.315} C_VEL
LIN {X 0,Y 294.971,Z 711.13,A -85,B 0,C 180,E1 -16759.485,E2 -16759.485} C_VEL
LIN {X 0,Y 296.185,Z 700.85,A -85,B 0,C 180,E1 -16761.579,E2 -16761.579} C_VEL
LIN {X 0,Y 297.509,Z 688.476,A -85,B 0,C 180,E1 -16763.677,E2 -16763.677} C_VEL
LIN {X 0,Y 298.773,Z 676.012,A -85,B 0,C 180,E1 -16765.422,E2 -16765.422} C_VEL
LIN {X 0,Y 300.046,Z 662.309,A -85,B 0,C 180,E1 -16766.996,E2 -16766.996} C_VEL
LIN {X 0,Y 301.14,Z 648.215,A -85,B 0,C 180,E1 -16768.297,E2 -16768.297} C_VEL
LIN {X 0,Y 302.053,Z 632.766,A -85,B 0,C 180,E1 -16769.411,E2 -16769.411} C_VEL
LIN {X 0,Y 302.806,Z 616.78,A -85,B 0,C 180,E1 -16770.256,E2 -16770.256} C_VEL
LIN {X 0,Y 303.109,Z 596.522,A -85,B 0,C 180,E1 -16771.002,E2 -16771.002} C_VEL
LIN {X 0,Y 291.397,Z 564.217,A -85,B 0,C 180,E1 -16772.842,E2 -16772.842} C_VEL
LIN {X 0,Y 291.382,Z 564.186,A -85,B 0,C 180,E1 -16777.254,E2 -16777.254} C_VEL
LIN {X 0,Y 291.334,Z 564.193,A -85,B 0,C 180,E1 -16780.641,E2 -16780.641} C_VEL
LIN {X 0,Y 291.291,Z 564.202,A -85,B 0,C 180,E1 -16784.401,E2 -16784.401} C_VEL
LIN {X 0,Y 291.347,Z 564.195,A -85,B 0,C 180,E1 -16788.399,E2 -16788.399} C_VEL
LIN {X 0,Y 291.365,Z 564.188,A -85,B 0,C 180,E1 -16791.159,E2 -16791.159} C_VEL
LIN {X 0,Y 291.385,Z 564.19,A -85,B 0,C 180,E1 -16794.629,E2 -16794.629} C_VEL
LIN {X 0,Y 291.37,Z 564.187,A -85,B 0,C 180,E1 -16797.95,E2 -16797.95} C_VEL
LIN {X 0,Y 291.376,Z 564.188,A -85,B 0,C 180,E1 -16801.157,E2 -16801.157} C_VEL
LIN {X 0,Y 291.412,Z 564.184,A -85,B 0,C 180,E1 -16804.271,E2 -16804.271} C_VEL
LIN {X 0,Y 291.381,Z 564.187,A -85,B 0,C 180,E1 -16807.299,E2 -16807.299} C_VEL
LIN {X 0,Y 291.457,Z 564.178,A -85,B 0,C 180,E1 -16810.269,E2 -16810.269} C_VEL
LIN {X 0,Y 291.554,Z 564.167,A -85,B 0,C 180,E1 -16814.623,E2 -16814.623} C_VEL
LIN {X 0,Y 291.535,Z 564.172,A -85,B 0,C 180,E1 -16818.88,E2 -16818.88} C_VEL
LIN {X 0,Y 291.707,Z 564.146,A -85,B 0,C 180,E1 -16821.688,E2 -16821.688} C_VEL
LIN {X 0,Y 291.63,Z 564.155,A -85,B 0,C 180,E1 -16824.468,E2 -16824.468} C_VEL
LIN {X 0,Y 291.888,Z 564.124,A -85,B 0,C 180,E1 -16828.62,E2 -16828.62} C_VEL
LIN {X 0,Y 291.888,Z 564.126,A -85,B 0,C 180,E1 -16831.379,E2 -16831.379} C_VEL
LIN {X 0,Y 291.743,Z 564.143,A -85,B 0,C 180,E1 -16836.917,E2 -16836.917} C_VEL
LIN {X 0,Y 291.627,Z 564.157,A -85,B 0,C 180,E1 -16839.711,E2 -16839.711} C_VEL
LIN {X 0,Y 291.52,Z 564.17,A -85,B 0,C 180,E1 -16843.949,E2 -16843.949} C_VEL
LIN {X 0,Y 291.484,Z 564.174,A -85,B 0,C 180,E1 -16846.817,E2 -16846.817} C_VEL
LIN {X 0,Y 291.447,Z 564.179,A -85,B 0,C 180,E1 -16849.874,E2 -16849.874} C_VEL
LIN {X 0,Y 291.396,Z 564.185,A -85,B 0,C 180,E1 -16854.205,E2 -16854.205} C_VEL
LIN {X 0,Y 291.418,Z 564.184,A -85,B 0,C 180,E1 -16857.271,E2 -16857.271} C_VEL
LIN {X 0,Y 291.335,Z 564.191,A -85,B 0,C 180,E1 -16860.436,E2 -16860.436} C_VEL
LIN {X 0,Y 291.341,Z 564.196,A -85,B 0,C 180,E1 -16863.698,E2 -16863.698} C_VEL
LIN {X 0,Y 291.399,Z 564.185,A -85,B 0,C 180,E1 -16867.261,E2 -16867.261} C_VEL
LIN {X 0,Y 291.373,Z 564.188,A -85,B 0,C 180,E1 -16870.634,E2 -16870.634} C_VEL
LIN {X 0,Y 291.391,Z 564.187,A -85,B 0,C 180,E1 -16874.381,E2 -16874.381} C_VEL
LIN {X 0,Y 291.385,Z 564.189,A -85,B 0,C 180,E1 -16878.39,E2 -16878.39} C_VEL
LIN {X 0,Y 291.431,Z 564.209,A -85,B 0,C 180,E1 -16879.702,E2 -16879.702} C_VEL
LIN {X 0,Y 302.012,Z 593.033,A -85,B 0,C 180,E1 -16881.307,E2 -16881.307} C_VEL
LIN {X 0,Y 301.259,Z 627.574,A -85,B 0,C 180,E1 -16882.411,E2 -16882.411} C_VEL
LIN {X 0,Y 300.768,Z 641.982,A -85,B 0,C 180,E1 -16883.114,E2 -16883.114} C_VEL
LIN {X 0,Y 300.08,Z 655.767,A -85,B 0,C 180,E1 -16884.058,E2 -16884.058} C_VEL
LIN {X 0,Y 299.133,Z 668.07,A -85,B 0,C 180,E1 -16885.144,E2 -16885.144} C_VEL
LIN {X 0,Y 298.048,Z 680.767,A -85,B 0,C 180,E1 -16886.552,E2 -16886.552} C_VEL
LIN {X 0,Y 296.805,Z 692.894,A -85,B 0,C 180,E1 -16888.208,E2 -16888.208} C_VEL
LIN {X 0,Y 295.69,Z 703.881,A -85,B 0,C 180,E1 -16890.058,E2 -16890.058} C_VEL
LIN {X 0,Y 294.609,Z 713.231,A -85,B 0,C 180,E1 -16891.961,E2 -16891.961} C_VEL
LIN {X 0,Y 293.623,Z 721.926,A -85,B 0,C 180,E1 -16894.099,E2 -16894.099} C_VEL
LIN {X 0,Y 292.874,Z 729.265,A -85,B 0,C 180,E1 -16896.301,E2 -16896.301} C_VEL
LIN {X 0,Y 292.195,Z 736.112,A -85,B 0,C 180,E1 -16898.852,E2 -16898.852} C_VEL
LIN {X 0,Y 291.73,Z 741.402,A -85,B 0,C 180,E1 -16901.449,E2 -16901.449} C_VEL
LIN {X 0,Y 290.951,Z 743.315,A -85,B 0,C 180,E1 -16902.539,E2 -16902.539} C_VEL
LIN {X 0,Y 288.049,Z 746.188,A -85,B 0,C 180,E1 -16904.328,E2 -16904.328} C_VEL
LIN {X 0,Y 285.7,Z 748.038,A -85,B 0,C 180,E1 -16905.802,E2 -16905.802} C_VEL
LIN {X 0,Y 284.757,Z 749.052,A -85,B 0,C 180,E1 -16906.96,E2 -16906.96} C_VEL
LIN {X 0,Y 284.712,Z 749.3,A -85,B 0,C 180,E1 -16907.354,E2 -16907.354} C_VEL
LIN {X 0,Y 285.189,Z 750.42,A -85,B 0,C 180,E1 -16910.067,E2 -16910.067} C_VEL
LIN {X 0,Y 285.969,Z 750.152,A -85,B 0,C 180,E1 -16912.942,E2 -16912.942} C_VEL
LIN {X 0,Y 287.215,Z 748.422,A -85,B 0,C 180,E1 -16915.791,E2 -16915.791} C_VEL
LIN {X 0,Y 288.35,Z 746.209,A -85,B 0,C 180,E1 -16917.826,E2 -16917.826} C_VEL
LIN {X 0,Y 289.767,Z 742.924,A -85,B 0,C 180,E1 -16920.001,E2 -16920.001} C_VEL
LIN {X 0,Y 292.005,Z 737.214,A -85,B 0,C 180,E1 -16922.76,E2 -16922.76} C_VEL
LIN {X 0,Y 294.229,Z 730.701,A -85,B 0,C 180,E1 -16925.14,E2 -16925.14} C_VEL
LIN {X 0,Y 296.519,Z 723.671,A -85,B 0,C 180,E1 -16927.149,E2 -16927.149} C_VEL
LIN {X 0,Y 299.044,Z 714.689,A -85,B 0,C 180,E1 -16929.232,E2 -16929.232} C_VEL
LIN {X 0,Y 301.36,Z 705.413,A -85,B 0,C 180,E1 -16930.999,E2 -16930.999} C_VEL
LIN {X 0,Y 303.649,Z 695.439,A -85,B 0,C 180,E1 -16932.533,E2 -16932.533} C_VEL
LIN {X 0,Y 305.738,Z 684.305,A -85,B 0,C 180,E1 -16933.941,E2 -16933.941} C_VEL
LIN {X 0,Y 307.67,Z 671.45,A -85,B 0,C 180,E1 -16935.23,E2 -16935.23} C_VEL
LIN {X 0,Y 309.134,Z 657.681,A -85,B 0,C 180,E1 -16936.325,E2 -16936.325} C_VEL
LIN {X 0,Y 310.095,Z 644.078,A -85,B 0,C 180,E1 -16937.106,E2 -16937.106} C_VEL
LIN {X 0,Y 310.782,Z 626.304,A -85,B 0,C 180,E1 -16937.816,E2 -16937.816} C_VEL
LIN {X 0,Y 311.793,Z 606.614,A -85,B 0,C 180,E1 -16938.528,E2 -16938.528} C_VEL
LIN {X 0,Y 306.928,Z 597.563,A -85,B 0,C 180,E1 -16940.01,E2 -16940.01} C_VEL
LIN {X 0,Y 302.135,Z 589.519,A -85,B 0,C 180,E1 -16941.636,E2 -16941.636} C_VEL
LIN {X 0,Y 298.883,Z 584.887,A -85,B 0,C 180,E1 -16942.828,E2 -16942.828} C_VEL
LIN {X 0,Y 295.974,Z 580.724,A -85,B 0,C 180,E1 -16944.014,E2 -16944.014} C_VEL
LIN {X 0,Y 293.355,Z 577.247,A -85,B 0,C 180,E1 -16945.176,E2 -16945.176} C_VEL
LIN {X 0,Y 292.649,Z 575.958,A -85,B 0,C 180,E1 -16945.549,E2 -16945.549} C_VEL
LIN {X 0,Y 290.189,Z 573.59,A -85,B 0,C 180,E1 -16946.741,E2 -16946.741} C_VEL
LIN {X 0,Y 288.821,Z 570.792,A -85,B 0,C 180,E1 -16947.644,E2 -16947.644} C_VEL
LIN {X 0,Y 286.035,Z 568.845,A -85,B 0,C 180,E1 -16949.315,E2 -16949.315} C_VEL
LIN {X 0,Y 284.537,Z 566.178,A -85,B 0,C 180,E1 -16950.593,E2 -16950.593} C_VEL
LIN {X 0,Y 284.279,Z 565.066,A -85,B 0,C 180,E1 -16950.95,E2 -16950.95} C_VEL
LIN {X 0,Y 284.307,Z 565.058,A -85,B 0,C 180,E1 -16954.65,E2 -16954.65} C_VEL
LIN {X 0,Y 284.317,Z 565.066,A -85,B 0,C 180,E1 -16958.169,E2 -16958.169} C_VEL
LIN {X 0,Y 284.268,Z 565.07,A -85,B 0,C 180,E1 -16962.125,E2 -16962.125} C_VEL
LIN {X 0,Y 284.3,Z 565.272,A -85,B 0,C 180,E1 -16965.635,E2 -16965.635} C_VEL
LIN {X 0,Y 285.118,Z 567.661,A -85,B 0,C 180,E1 -16966.564,E2 -16966.564} C_VEL
LIN {X 0,Y 286.987,Z 569.805,A -85,B 0,C 180,E1 -16967.906,E2 -16967.906} C_VEL
LIN {X 0,Y 288.864,Z 570.985,A -85,B 0,C 180,E1 -16968.996,E2 -16968.996} C_VEL
LIN {X 0,Y 292.076,Z 582.212,A -85,B 0,C 180,E1 -16971.408,E2 -16971.408} C_VEL
LIN {X 0,Y 294.307,Z 587.625,A -85,B 0,C 180,E1 -16972.646,E2 -16972.646} C_VEL
LIN {X 0,Y 296.593,Z 595.402,A -85,B 0,C 180,E1 -16973.951,E2 -16973.951} C_VEL
LIN {X 0,Y 297.962,Z 599.022,A -85,B 0,C 180,E1 -16974.605,E2 -16974.605} C_VEL
LIN {X 0,Y 299.05,Z 606.039,A -85,B 0,C 180,E1 -16975.375,E2 -16975.375} C_VEL
LIN {X 0,Y 300.789,Z 617.809,A -85,B 0,C 180,E1 -16976.564,E2 -16976.564} C_VEL
LIN {X 0,Y 303.041,Z 635.939,A -85,B 0,C 180,E1 -16978.146,E2 -16978.146} C_VEL
LIN {X 0,Y 304.83,Z 655.128,A -85,B 0,C 180,E1 -16979.561,E2 -16979.561} C_VEL
LIN {X 0,Y 306.037,Z 689.233,A -85,B 0,C 180,E1 -16981.5,E2 -16981.5} C_VEL
LIN {X 0,Y 304.07,Z 713.588,A -85,B 0,C 180,E1 -16982.419,E2 -16982.419} C_VEL
LIN {X 0,Y 302.055,Z 728.516,A -85,B 0,C 180,E1 -16983.206,E2 -16983.206} C_VEL
LIN {X 0,Y 299.75,Z 741.47,A -85,B 0,C 180,E1 -16984.108,E2 -16984.108} C_VEL
LIN {X 0,Y 296.983,Z 755.111,A -85,B 0,C 180,E1 -16985.35,E2 -16985.35} C_VEL
LIN {X 0,Y 293.929,Z 768.607,A -85,B 0,C 180,E1 -16986.951,E2 -16986.951} C_VEL
LIN {X 0,Y 291.499,Z 778.737,A -85,B 0,C 180,E1 -16988.429,E2 -16988.429} C_VEL
LIN {X 0,Y 289.149,Z 788.217,A -85,B 0,C 180,E1 -16990.107,E2 -16990.107} C_VEL
LIN {X 0,Y 286.968,Z 797.676,A -85,B 0,C 180,E1 -16992.175,E2 -16992.175} C_VEL
LIN {X 0,Y 285.325,Z 805.573,A -85,B 0,C 180,E1 -16994.28,E2 -16994.28} C_VEL
LIN {X 0,Y 284.204,Z 812.072,A -85,B 0,C 180,E1 -16996.414,E2 -16996.414} C_VEL
LIN {X 0,Y 283.46,Z 817.375,A -85,B 0,C 180,E1 -16998.56,E2 -16998.56} C_VEL
LIN {X 0,Y 283.269,Z 821.6,A -85,B 0,C 180,E1 -17000.72,E2 -17000.72} C_VEL
LIN {X 0,Y 283.398,Z 824.798,A -85,B 0,C 180,E1 -17002.878,E2 -17002.878} C_VEL
LIN {X 0,Y 283.624,Z 826.373,A -85,B 0,C 180,E1 -17004.313,E2 -17004.313} C_VEL
LIN {X 0,Y 283.939,Z 827.526,A -85,B 0,C 180,E1 -17005.742,E2 -17005.742} C_VEL
LIN {X 0,Y 284.51,Z 828.702,A -85,B 0,C 180,E1 -17008.585,E2 -17008.585} C_VEL
LIN {X 0,Y 284.683,Z 829.622,A -85,B 0,C 180,E1 -17010.001,E2 -17010.001} C_VEL
LIN {X 0,Y 284.275,Z 829.962,A -85,B 0,C 180,E1 -17011.417,E2 -17011.417} C_VEL
LIN {X 0,Y 283.94,Z 829.828,A -85,B 0,C 180,E1 -17012.838,E2 -17012.838} C_VEL
LIN {X 0,Y 283.761,Z 829.267,A -85,B 0,C 180,E1 -17014.262,E2 -17014.262} C_VEL
LIN {X 0,Y 283.26,Z 826.893,A -85,B 0,C 180,E1 -17017.043,E2 -17017.043} C_VEL
LIN {X 0,Y 283.112,Z 823.808,A -85,B 0,C 180,E1 -17019.286,E2 -17019.286} C_VEL
LIN {X 0,Y 283.345,Z 819.848,A -85,B 0,C 180,E1 -17021.446,E2 -17021.446} C_VEL
LIN {X 0,Y 284.111,Z 814.886,A -85,B 0,C 180,E1 -17023.592,E2 -17023.592} C_VEL
LIN {X 0,Y 285.405,Z 807.331,A -85,B 0,C 180,E1 -17026.184,E2 -17026.184} C_VEL
LIN {X 0,Y 287.628,Z 798.76,A -85,B 0,C 180,E1 -17028.521,E2 -17028.521} C_VEL
LIN {X 0,Y 290.188,Z 789.592,A -85,B 0,C 180,E1 -17030.56,E2 -17030.56} C_VEL
LIN {X 0,Y 293.262,Z 778.7,A -85,B 0,C 180,E1 -17032.548,E2 -17032.548} C_VEL
LIN {X 0,Y 296.545,Z 766.763,A -85,B 0,C 180,E1 -17034.318,E2 -17034.318} C_VEL
LIN {X 0,Y 300.493,Z 752.4,A -85,B 0,C 180,E1 -17036.011,E2 -17036.011} C_VEL
LIN {X 0,Y 304.073,Z 737.992,A -85,B 0,C 180,E1 -17037.347,E2 -17037.347} C_VEL
LIN {X 0,Y 307.461,Z 722.313,A -85,B 0,C 180,E1 -17038.501,E2 -17038.501} C_VEL
LIN {X 0,Y 310.651,Z 704.35,A -85,B 0,C 180,E1 -17039.477,E2 -17039.477} C_VEL
LIN {X 0,Y 312.481,Z 687.935,A -85,B 0,C 180,E1 -17040.198,E2 -17040.198} C_VEL
LIN {X 0,Y 313.605,Z 661.924,A -85,B 0,C 180,E1 -17041.571,E2 -17041.571} C_VEL
LIN {X 0,Y 313.675,Z 646.082,A -85,B 0,C 180,E1 -17042.631,E2 -17042.631} C_VEL
LIN {X 0,Y 313.057,Z 629.783,A -85,B 0,C 180,E1 -17044.011,E2 -17044.011} C_VEL
LIN {X 0,Y 312.103,Z 614.718,A -85,B 0,C 180,E1 -17045.578,E2 -17045.578} C_VEL
LIN {X 0,Y 311.229,Z 602.891,A -85,B 0,C 180,E1 -17047.043,E2 -17047.043} C_VEL
LIN {X 0,Y 309.953,Z 596.734,A -85,B 0,C 180,E1 -17048.328,E2 -17048.328} C_VEL
LIN {X 0,Y 308.495,Z 593.911,A -85,B 0,C 180,E1 -17049.508,E2 -17049.508} C_VEL
LIN {X 0,Y 306.15,Z 591.037,A -85,B 0,C 180,E1 -17051.805,E2 -17051.805} C_VEL
LIN {X 0,Y 305.478,Z 588.99,A -85,B 0,C 180,E1 -17053.136,E2 -17053.136} C_VEL
LIN {X 0,Y 304.69,Z 588.642,A -85,B 0,C 180,E1 -17056.212,E2 -17056.212} C_VEL
LIN {X 0,Y 305.777,Z 589.174,A -85,B 0,C 180,E1 -17058.923,E2 -17058.923} C_VEL
LIN {X 0,Y 306.965,Z 592.141,A -85,B 0,C 180,E1 -17060.697,E2 -17060.697} C_VEL
LIN {X 0,Y 309.023,Z 594.274,A -85,B 0,C 180,E1 -17062.332,E2 -17062.332} C_VEL
LIN {X 0,Y 311.124,Z 597.746,A -85,B 0,C 180,E1 -17063.793,E2 -17063.793} C_VEL
LIN {X 0,Y 314.098,Z 602.421,A -85,B 0,C 180,E1 -17065.42,E2 -17065.42} C_VEL
LIN {X 0,Y 316.841,Z 607.231,A -85,B 0,C 180,E1 -17066.716,E2 -17066.716} C_VEL
LIN {X 0,Y 320.075,Z 613.468,A -85,B 0,C 180,E1 -17068.065,E2 -17068.065} C_VEL
LIN {X 0,Y 318.673,Z 638.599,A -85,B 0,C 180,E1 -17069.154,E2 -17069.154} C_VEL
LIN {X 0,Y 317.4,Z 652.843,A -85,B 0,C 180,E1 -17070.026,E2 -17070.026} C_VEL
LIN {X 0,Y 315.805,Z 665.435,A -85,B 0,C 180,E1 -17070.998,E2 -17070.998} C_VEL
LIN {X 0,Y 313.733,Z 677.306,A -85,B 0,C 180,E1 -17072.119,E2 -17072.119} C_VEL
LIN {X 0,Y 311.291,Z 689.139,A -85,B 0,C 180,E1 -17073.519,E2 -17073.519} C_VEL
LIN {X 0,Y 308.583,Z 700.17,A -85,B 0,C 180,E1 -17075.08,E2 -17075.08} C_VEL
LIN {X 0,Y 305.915,Z 709.516,A -85,B 0,C 180,E1 -17076.689,E2 -17076.689} C_VEL
LIN {X 0,Y 302.86,Z 719.252,A -85,B 0,C 180,E1 -17078.718,E2 -17078.718} C_VEL
LIN {X 0,Y 299.806,Z 727.648,A -85,B 0,C 180,E1 -17080.841,E2 -17080.841} C_VEL
LIN {X 0,Y 297.272,Z 733.943,A -85,B 0,C 180,E1 -17082.811,E2 -17082.811} C_VEL
LIN {X 0,Y 294.266,Z 740.85,A -85,B 0,C 180,E1 -17085.476,E2 -17085.476} C_VEL
LIN {X 0,Y 291.661,Z 746.103,A -85,B 0,C 180,E1 -17088.18,E2 -17088.18} C_VEL
LIN {X 0,Y 289.994,Z 749.024,A -85,B 0,C 180,E1 -17090.232,E2 -17090.232} C_VEL
LIN {X 0,Y 288.339,Z 751.78,A -85,B 0,C 180,E1 -17092.999,E2 -17092.999} C_VEL
LIN {X 0,Y 286.875,Z 753.289,A -85,B 0,C 180,E1 -17095.785,E2 -17095.785} C_VEL
LIN {X 0,Y 285.888,Z 753.516,A -85,B 0,C 180,E1 -17098.591,E2 -17098.591} C_VEL
LIN {X 0,Y 285.219,Z 752.505,A -85,B 0,C 180,E1 -17101.411,E2 -17101.411} C_VEL
LIN {X 0,Y 284.764,Z 750.25,A -85,B 0,C 180,E1 -17104.245,E2 -17104.245} C_VEL
LIN {X 0,Y 284.851,Z 746.662,A -85,B 0,C 180,E1 -17107.086,E2 -17107.086} C_VEL
LIN {X 0,Y 285.021,Z 741.701,A -85,B 0,C 180,E1 -17109.939,E2 -17109.939} C_VEL
LIN {X 0,Y 285.476,Z 735.213,A -85,B 0,C 180,E1 -17112.8,E2 -17112.8} C_VEL
LIN {X 0,Y 286.172,Z 728.087,A -85,B 0,C 180,E1 -17115.307,E2 -17115.307} C_VEL
LIN {X 0,Y 287.136,Z 719.393,A -85,B 0,C 180,E1 -17117.815,E2 -17117.815} C_VEL
LIN {X 0,Y 288.274,Z 708.748,A -85,B 0,C 180,E1 -17120.328,E2 -17120.328} C_VEL
LIN {X 0,Y 289.602,Z 697.74,A -85,B 0,C 180,E1 -17122.47,E2 -17122.47} C_VEL
LIN {X 0,Y 290.897,Z 685.601,A -85,B 0,C 180,E1 -17124.439,E2 -17124.439} C_VEL
LIN {X 0,Y 292.334,Z 672.291,A -85,B 0,C 180,E1 -17126.215,E2 -17126.215} C_VEL
LIN {X 0,Y 293.519,Z 658.239,A -85,B 0,C 180,E1 -17127.749,E2 -17127.749} C_VEL
LIN {X 0,Y 294.523,Z 643.984,A -85,B 0,C 180,E1 -17128.992,E2 -17128.992} C_VEL
LIN {X 0,Y 295.408,Z 628.901,A -85,B 0,C 180,E1 -17130.002,E2 -17130.002} C_VEL
LIN {X 0,Y 295.996,Z 613.649,A -85,B 0,C 180,E1 -17130.745,E2 -17130.745} C_VEL
LIN {X 0,Y 296.179,Z 597.743,A -85,B 0,C 180,E1 -17131.323,E2 -17131.323} C_VEL
LIN {X 0,Y 284.344,Z 565.063,A -85,B 0,C 180,E1 -17133.288,E2 -17133.288} C_VEL
LIN {X 0,Y 284.335,Z 565.067,A -85,B 0,C 180,E1 -17136.385,E2 -17136.385} C_VEL
LIN {X 0,Y 284.307,Z 565.071,A -85,B 0,C 180,E1 -17139.994,E2 -17139.994} C_VEL
LIN {X 0,Y 284.246,Z 565.079,A -85,B 0,C 180,E1 -17144.19,E2 -17144.19} C_VEL
LIN {X 0,Y 284.289,Z 565.072,A -85,B 0,C 180,E1 -17148.127,E2 -17148.127} C_VEL
LIN {X 0,Y 284.335,Z 565.067,A -85,B 0,C 180,E1 -17152.274,E2 -17152.274} C_VEL
LIN {X 0,Y 284.323,Z 565.065,A -85,B 0,C 180,E1 -17155.352,E2 -17155.352} C_VEL
LIN {X 0,Y 284.293,Z 565.073,A -85,B 0,C 180,E1 -17158.725,E2 -17158.725} C_VEL
LIN {X 0,Y 284.393,Z 565.06,A -85,B 0,C 180,E1 -17162.827,E2 -17162.827} C_VEL
LIN {X 0,Y 284.366,Z 565.064,A -85,B 0,C 180,E1 -17166.706,E2 -17166.706} C_VEL
LIN {X 0,Y 284.402,Z 565.057,A -85,B 0,C 180,E1 -17171.261,E2 -17171.261} C_VEL
LIN {X 0,Y 284.491,Z 565.046,A -85,B 0,C 180,E1 -17174.458,E2 -17174.458} C_VEL
LIN {X 0,Y 284.487,Z 565.047,A -85,B 0,C 180,E1 -17178.601,E2 -17178.601} C_VEL
LIN {X 0,Y 284.657,Z 565.025,A -85,B 0,C 180,E1 -17181.48,E2 -17181.48} C_VEL
LIN {X 0,Y 284.6,Z 565.03,A -85,B 0,C 180,E1 -17184.33,E2 -17184.33} C_VEL
LIN {X 0,Y 284.854,Z 565,A -85,B 0,C 180,E1 -17188.585,E2 -17188.585} C_VEL
LIN {X 0,Y 284.854,Z 565.002,A -85,B 0,C 180,E1 -17191.413,E2 -17191.413} C_VEL
LIN {X 0,Y 284.695,Z 565.023,A -85,B 0,C 180,E1 -17197.089,E2 -17197.089} C_VEL
LIN {X 0,Y 284.564,Z 565.036,A -85,B 0,C 180,E1 -17199.955,E2 -17199.955} C_VEL
LIN {X 0,Y 284.479,Z 565.046,A -85,B 0,C 180,E1 -17204.302,E2 -17204.302} C_VEL
LIN {X 0,Y 284.422,Z 565.057,A -85,B 0,C 180,E1 -17207.248,E2 -17207.248} C_VEL
LIN {X 0,Y 284.376,Z 565.058,A -85,B 0,C 180,E1 -17210.241,E2 -17210.241} C_VEL
LIN {X 0,Y 284.365,Z 565.063,A -85,B 0,C 180,E1 -17213.875,E2 -17213.875} C_VEL
LIN {X 0,Y 284.393,Z 565.058,A -85,B 0,C 180,E1 -17217.173,E2 -17217.173} C_VEL
LIN {X 0,Y 284.294,Z 565.07,A -85,B 0,C 180,E1 -17221.273,E2 -17221.273} C_VEL
LIN {X 0,Y 284.357,Z 565.063,A -85,B 0,C 180,E1 -17225.354,E2 -17225.354} C_VEL
LIN {X 0,Y 284.329,Z 565.067,A -85,B 0,C 180,E1 -17228.165,E2 -17228.165} C_VEL
LIN {X 0,Y 284.312,Z 565.07,A -85,B 0,C 180,E1 -17232.135,E2 -17232.135} C_VEL
LIN {X 0,Y 284.344,Z 565.067,A -85,B 0,C 180,E1 -17236.207,E2 -17236.207} C_VEL
LIN {X 0,Y 284.384,Z 565.059,A -85,B 0,C 180,E1 -17239.247,E2 -17239.247} C_VEL
LIN {X 0,Y 295.157,Z 594.605,A -85,B 0,C 180,E1 -17240.96,E2 -17240.96} C_VEL
LIN {X 0,Y 294.37,Z 629.272,A -85,B 0,C 180,E1 -17242.107,E2 -17242.107} C_VEL
LIN {X 0,Y 293.85,Z 643.933,A -85,B 0,C 180,E1 -17242.853,E2 -17242.853} C_VEL
LIN {X 0,Y 293.014,Z 658.503,A -85,B 0,C 180,E1 -17243.905,E2 -17243.905} C_VEL
LIN {X 0,Y 292.044,Z 671.661,A -85,B 0,C 180,E1 -17245.143,E2 -17245.143} C_VEL
LIN {X 0,Y 290.87,Z 684.483,A -85,B 0,C 180,E1 -17246.655,E2 -17246.655} C_VEL
LIN {X 0,Y 289.59,Z 696.385,A -85,B 0,C 180,E1 -17248.403,E2 -17248.403} C_VEL
LIN {X 0,Y 288.351,Z 707.609,A -85,B 0,C 180,E1 -17250.426,E2 -17250.426} C_VEL
LIN {X 0,Y 287.366,Z 716.256,A -85,B 0,C 180,E1 -17252.312,E2 -17252.312} C_VEL
LIN {X 0,Y 286.389,Z 724.859,A -85,B 0,C 180,E1 -17254.568,E2 -17254.568} C_VEL
LIN {X 0,Y 285.624,Z 731.84,A -85,B 0,C 180,E1 -17256.816,E2 -17256.816} C_VEL
LIN {X 0,Y 284.973,Z 738.627,A -85,B 0,C 180,E1 -17259.576,E2 -17259.576} C_VEL
LIN {X 0,Y 284.628,Z 743.256,A -85,B 0,C 180,E1 -17262.023,E2 -17262.023} C_VEL
LIN {X 0,Y 284.52,Z 746.647,A -85,B 0,C 180,E1 -17264.436,E2 -17264.436} C_VEL
LIN {X 0,Y 284.712,Z 749.3,A -85,B 0,C 180,E1 -17267.354,E2 -17267.354} C_VEL
LIN {X 0,Y 284.197,Z 750.068,A -85,B 0,C 180,E1 -17268.532,E2 -17268.532} C_VEL
LIN {X 0,Y 281.723,Z 751.029,A -85,B 0,C 180,E1 -17270.467,E2 -17270.467} C_VEL
LIN {X 0,Y 279.763,Z 751.43,A -85,B 0,C 180,E1 -17272.039,E2 -17272.039} C_VEL
LIN {X 0,Y 279.166,Z 751.352,A -85,B 0,C 180,E1 -17273.247,E2 -17273.247} C_VEL
LIN {X 0,Y 279.249,Z 751.199,A -85,B 0,C 180,E1 -17273.651,E2 -17273.651} C_VEL
LIN {X 0,Y 280.176,Z 750.074,A -85,B 0,C 180,E1 -17275.685,E2 -17275.685} C_VEL
LIN {X 0,Y 281.839,Z 747.153,A -85,B 0,C 180,E1 -17278.572,E2 -17278.572} C_VEL
LIN {X 0,Y 283.378,Z 743.932,A -85,B 0,C 180,E1 -17280.711,E2 -17280.711} C_VEL
LIN {X 0,Y 285.166,Z 739.764,A -85,B 0,C 180,E1 -17282.826,E2 -17282.826} C_VEL
LIN {X 0,Y 287.113,Z 734.578,A -85,B 0,C 180,E1 -17284.915,E2 -17284.915} C_VEL
LIN {X 0,Y 289.797,Z 726.99,A -85,B 0,C 180,E1 -17287.315,E2 -17287.315} C_VEL
LIN {X 0,Y 292.519,Z 718.549,A -85,B 0,C 180,E1 -17289.44,E2 -17289.44} C_VEL
LIN {X 0,Y 294.921,Z 709.783,A -85,B 0,C 180,E1 -17291.242,E2 -17291.242} C_VEL
LIN {X 0,Y 297.524,Z 699.308,A -85,B 0,C 180,E1 -17292.969,E2 -17292.969} C_VEL
LIN {X 0,Y 299.997,Z 687.34,A -85,B 0,C 180,E1 -17294.587,E2 -17294.587} C_VEL
LIN {X 0,Y 302.101,Z 675.293,A -85,B 0,C 180,E1 -17295.864,E2 -17295.864} C_VEL
LIN {X 0,Y 303.729,Z 661.623,A -85,B 0,C 180,E1 -17297.01,E2 -17297.01} C_VEL
LIN {X 0,Y 304.927,Z 647.554,A -85,B 0,C 180,E1 -17297.89,E2 -17297.89} C_VEL
LIN {X 0,Y 305.76,Z 629.123,A -85,B 0,C 180,E1 -17298.686,E2 -17298.686} C_VEL
LIN {X 0,Y 306.926,Z 609.754,A -85,B 0,C 180,E1 -17299.393,E2 -17299.393} C_VEL
LIN {X 0,Y 302.514,Z 601.329,A -85,B 0,C 180,E1 -17300.866,E2 -17300.866} C_VEL
LIN {X 0,Y 298.474,Z 594.698,A -85,B 0,C 180,E1 -17302.319,E2 -17302.319} C_VEL
LIN {X 0,Y 295.43,Z 590.179,A -85,B 0,C 180,E1 -17303.515,E2 -17303.515} C_VEL
LIN {X 0,Y 293,Z 586.576,A -85,B 0,C 180,E1 -17304.583,E2 -17304.583} C_VEL
LIN {X 0,Y 290.555,Z 583.023,A -85,B 0,C 180,E1 -17305.768,E2 -17305.768} C_VEL
LIN {X 0,Y 289.412,Z 581.758,A -85,B 0,C 180,E1 -17306.336,E2 -17306.336} C_VEL
LIN {X 0,Y 287.303,Z 578.929,A -85,B 0,C 180,E1 -17307.537,E2 -17307.537} C_VEL
LIN {X 0,Y 286.607,Z 577.446,A -85,B 0,C 180,E1 -17308.024,E2 -17308.024} C_VEL
LIN {X 0,Y 283.738,Z 575.029,A -85,B 0,C 180,E1 -17309.899,E2 -17309.899} C_VEL
LIN {X 0,Y 282.358,Z 571.986,A -85,B 0,C 180,E1 -17311.305,E2 -17311.305} C_VEL
LIN {X 0,Y 279.294,Z 570.07,A -85,B 0,C 180,E1 -17314.923,E2 -17314.923} C_VEL
LIN {X 0,Y 278.551,Z 569.168,A -85,B 0,C 180,E1 -17317.268,E2 -17317.268} C_VEL
LIN {X 0,Y 278.724,Z 569.424,A -85,B 0,C 180,E1 -17320.111,E2 -17320.111} C_VEL
LIN {X 0,Y 280.936,Z 571.318,A -85,B 0,C 180,E1 -17323.917,E2 -17323.917} C_VEL
LIN {X 0,Y 282.323,Z 572.108,A -85,B 0,C 180,E1 -17325.256,E2 -17325.256} C_VEL
LIN {X 0,Y 283.714,Z 575.144,A -85,B 0,C 180,E1 -17326.691,E2 -17326.691} C_VEL
LIN {X 0,Y 286.349,Z 577.445,A -85,B 0,C 180,E1 -17328.466,E2 -17328.466} C_VEL
LIN {X 0,Y 289.365,Z 588.364,A -85,B 0,C 180,E1 -17330.899,E2 -17330.899} C_VEL
LIN {X 0,Y 290.986,Z 592.759,A -85,B 0,C 180,E1 -17331.902,E2 -17331.902} C_VEL
LIN {X 0,Y 293.15,Z 600.47,A -85,B 0,C 180,E1 -17333.254,E2 -17333.254} C_VEL
LIN {X 0,Y 294.131,Z 603.299,A -85,B 0,C 180,E1 -17333.771,E2 -17333.771} C_VEL
LIN {X 0,Y 295.781,Z 615.343,A -85,B 0,C 180,E1 -17335.105,E2 -17335.105} C_VEL
LIN {X 0,Y 297.826,Z 632.873,A -85,B 0,C 180,E1 -17336.768,E2 -17336.768} C_VEL
LIN {X 0,Y 299.628,Z 652.873,A -85,B 0,C 180,E1 -17338.365,E2 -17338.365} C_VEL
LIN {X 0,Y 299.961,Z 661.371,A -85,B 0,C 180,E1 -17338.922,E2 -17338.922} C_VEL
LIN {X 0,Y 300.778,Z 690.255,A -85,B 0,C 180,E1 -17340.615,E2 -17340.615} C_VEL
LIN {X 0,Y 298.661,Z 713.875,A -85,B 0,C 180,E1 -17341.547,E2 -17341.547} C_VEL
LIN {X 0,Y 296.45,Z 728.648,A -85,B 0,C 180,E1 -17342.37,E2 -17342.37} C_VEL
LIN {X 0,Y 293.851,Z 742.099,A -85,B 0,C 180,E1 -17343.357,E2 -17343.357} C_VEL
LIN {X 0,Y 290.646,Z 756.577,A -85,B 0,C 180,E1 -17344.775,E2 -17344.775} C_VEL
LIN {X 0,Y 287.752,Z 768.413,A -85,B 0,C 180,E1 -17346.236,E2 -17346.236} C_VEL
LIN {X 0,Y 285.438,Z 777.238,A -85,B 0,C 180,E1 -17347.566,E2 -17347.566} C_VEL
LIN {X 0,Y 282.962,Z 786.682,A -85,B 0,C 180,E1 -17349.273,E2 -17349.273} C_VEL
LIN {X 0,Y 280.548,Z 796.194,A -85,B 0,C 180,E1 -17351.374,E2 -17351.374} C_VEL
LIN {X 0,Y 278.385,Z 805.252,A -85,B 0,C 180,E1 -17353.878,E2 -17353.878} C_VEL
LIN {X 0,Y 277.244,Z 811.6,A -85,B 0,C 180,E1 -17356.066,E2 -17356.066} C_VEL
LIN {X 0,Y 276.434,Z 816.749,A -85,B 0,C 180,E1 -17358.266,E2 -17358.266} C_VEL
LIN {X 0,Y 276.189,Z 820.826,A -85,B 0,C 180,E1 -17360.48,E2 -17360.48} C_VEL
LIN {X 0,Y 276.307,Z 823.966,A -85,B 0,C 180,E1 -17362.745,E2 -17362.745} C_VEL
LIN {X 0,Y 276.522,Z 825.428,A -85,B 0,C 180,E1 -17364.166,E2 -17364.166} C_VEL
LIN {X 0,Y 276.87,Z 826.518,A -85,B 0,C 180,E1 -17365.634,E2 -17365.634} C_VEL
LIN {X 0,Y 277.15,Z 827.122,A -85,B 0,C 180,E1 -17367.094,E2 -17367.094} C_VEL
LIN {X 0,Y 277.528,Z 827.325,A -85,B 0,C 180,E1 -17368.55,E2 -17368.55} C_VEL
LIN {X 0,Y 277.705,Z 828.31,A -85,B 0,C 180,E1 -17370.001,E2 -17370.001} C_VEL
LIN {X 0,Y 277.274,Z 828.718,A -85,B 0,C 180,E1 -17371.453,E2 -17371.453} C_VEL
LIN {X 0,Y 276.907,Z 828.688,A -85,B 0,C 180,E1 -17372.91,E2 -17372.91} C_VEL
LIN {X 0,Y 276.7,Z 828.213,A -85,B 0,C 180,E1 -17374.371,E2 -17374.371} C_VEL
LIN {X 0,Y 276.171,Z 825.886,A -85,B 0,C 180,E1 -17377.311,E2 -17377.311} C_VEL
LIN {X 0,Y 276.095,Z 821.885,A -85,B 0,C 180,E1 -17380.265,E2 -17380.265} C_VEL
LIN {X 0,Y 276.565,Z 817.751,A -85,B 0,C 180,E1 -17382.475,E2 -17382.475} C_VEL
LIN {X 0,Y 277.453,Z 812.605,A -85,B 0,C 180,E1 -17384.674,E2 -17384.674} C_VEL
LIN {X 0,Y 278.797,Z 806.38,A -85,B 0,C 180,E1 -17386.852,E2 -17386.852} C_VEL
LIN {X 0,Y 281.289,Z 797.551,A -85,B 0,C 180,E1 -17389.333,E2 -17389.333} C_VEL
LIN {X 0,Y 284.032,Z 788.482,A -85,B 0,C 180,E1 -17391.407,E2 -17391.407} C_VEL
LIN {X 0,Y 287.395,Z 777.729,A -85,B 0,C 180,E1 -17393.415,E2 -17393.415} C_VEL
LIN {X 0,Y 290.884,Z 766.044,A -85,B 0,C 180,E1 -17395.204,E2 -17395.204} C_VEL
LIN {X 0,Y 295.031,Z 751.968,A -85,B 0,C 180,E1 -17396.912,E2 -17396.912} C_VEL
LIN {X 0,Y 298.775,Z 738.079,A -85,B 0,C 180,E1 -17398.256,E2 -17398.256} C_VEL
LIN {X 0,Y 302.58,Z 721.878,A -85,B 0,C 180,E1 -17399.481,E2 -17399.481} C_VEL
LIN {X 0,Y 305.846,Z 705.361,A -85,B 0,C 180,E1 -17400.425,E2 -17400.425} C_VEL
LIN {X 0,Y 307.983,Z 689.2,A -85,B 0,C 180,E1 -17401.186,E2 -17401.186} C_VEL
LIN {X 0,Y 309.403,Z 663.644,A -85,B 0,C 180,E1 -17402.57,E2 -17402.57} C_VEL
LIN {X 0,Y 309.663,Z 648.201,A -85,B 0,C 180,E1 -17403.644,E2 -17403.644} C_VEL
LIN {X 0,Y 309.408,Z 633.703,A -85,B 0,C 180,E1 -17404.9,E2 -17404.9} C_VEL
LIN {X 0,Y 308.86,Z 619.16,A -85,B 0,C 180,E1 -17406.428,E2 -17406.428} C_VEL
LIN {X 0,Y 308.317,Z 607.477,A -85,B 0,C 180,E1 -17407.898,E2 -17407.898} C_VEL
LIN {X 0,Y 307.475,Z 602.652,A -85,B 0,C 180,E1 -17408.936,E2 -17408.936} C_VEL
LIN {X 0,Y 306.325,Z 600.394,A -85,B 0,C 180,E1 -17409.972,E2 -17409.972} C_VEL
LIN {X 0,Y 304.258,Z 597.354,A -85,B 0,C 180,E1 -17412.339,E2 -17412.339} C_VEL
LIN {X 0,Y 303.864,Z 595.886,A -85,B 0,C 180,E1 -17413.322,E2 -17413.322} C_VEL
LIN {X 0,Y 303.187,Z 595.591,A -85,B 0,C 180,E1 -17415.939,E2 -17415.939} C_VEL
LIN {X 0,Y 304.16,Z 596.108,A -85,B 0,C 180,E1 -17418.715,E2 -17418.715} C_VEL
LIN {X 0,Y 305.455,Z 599.218,A -85,B 0,C 180,E1 -17420.681,E2 -17420.681} C_VEL
LIN {X 0,Y 307.059,Z 600.961,A -85,B 0,C 180,E1 -17422.009,E2 -17422.009} C_VEL
LIN {X 0,Y 309.621,Z 605.291,A -85,B 0,C 180,E1 -17423.83,E2 -17423.83} C_VEL
LIN {X 0,Y 312.165,Z 609.702,A -85,B 0,C 180,E1 -17425.278,E2 -17425.278} C_VEL
LIN {X 0,Y 315.017,Z 615.094,A -85,B 0,C 180,E1 -17426.675,E2 -17426.675} C_VEL
LIN {X 0,Y 316.066,Z 617.441,A -85,B 0,C 180,E1 -17427.143,E2 -17427.143} C_VEL
LIN {X 0,Y 314.44,Z 640.428,A -85,B 0,C 180,E1 -17428.174,E2 -17428.174} C_VEL
LIN {X 0,Y 313.129,Z 654.451,A -85,B 0,C 180,E1 -17429.043,E2 -17429.043} C_VEL
LIN {X 0,Y 311.584,Z 665.69,A -85,B 0,C 180,E1 -17429.922,E2 -17429.922} C_VEL
LIN {X 0,Y 309.204,Z 678.316,A -85,B 0,C 180,E1 -17431.118,E2 -17431.118} C_VEL
LIN {X 0,Y 306.599,Z 690.276,A -85,B 0,C 180,E1 -17432.527,E2 -17432.527} C_VEL
LIN {X 0,Y 303.707,Z 701.197,A -85,B 0,C 180,E1 -17434.101,E2 -17434.101} C_VEL
LIN {X 0,Y 300.619,Z 711.295,A -85,B 0,C 180,E1 -17435.849,E2 -17435.849} C_VEL
LIN {X 0,Y 297.492,Z 720.471,A -85,B 0,C 180,E1 -17437.79,E2 -17437.79} C_VEL
LIN {X 0,Y 294.043,Z 729.328,A -85,B 0,C 180,E1 -17440.086,E2 -17440.086} C_VEL
LIN {X 0,Y 290.925,Z 736.573,A -85,B 0,C 180,E1 -17442.424,E2 -17442.424} C_VEL
LIN {X 0,Y 287.745,Z 743.089,A -85,B 0,C 180,E1 -17445.139,E2 -17445.139} C_VEL
LIN {X 0,Y 284.996,Z 748.083,A -85,B 0,C 180,E1 -17447.9,E2 -17447.9} C_VEL
LIN {X 0,Y 283.249,Z 750.896,A -85,B 0,C 180,E1 -17449.997,E2 -17449.997} C_VEL
LIN {X 0,Y 281.476,Z 753.399,A -85,B 0,C 180,E1 -17452.828,E2 -17452.828} C_VEL
LIN {X 0,Y 279.958,Z 754.692,A -85,B 0,C 180,E1 -17455.68,E2 -17455.68} C_VEL
LIN {X 0,Y 278.89,Z 754.72,A -85,B 0,C 180,E1 -17458.555,E2 -17458.555} C_VEL
LIN {X 0,Y 278.197,Z 753.493,A -85,B 0,C 180,E1 -17461.447,E2 -17461.447} C_VEL
LIN {X 0,Y 277.709,Z 751.029,A -85,B 0,C 180,E1 -17464.353,E2 -17464.353} C_VEL
LIN {X 0,Y 277.817,Z 747.219,A -85,B 0,C 180,E1 -17467.266,E2 -17467.266} C_VEL
LIN {X 0,Y 277.997,Z 742.015,A -85,B 0,C 180,E1 -17470.192,E2 -17470.192} C_VEL
LIN {X 0,Y 278.457,Z 735.214,A -85,B 0,C 180,E1 -17473.129,E2 -17473.129} C_VEL
LIN {X 0,Y 279.251,Z 727.805,A -85,B 0,C 180,E1 -17475.696,E2 -17475.696} C_VEL
LIN {X 0,Y 280.21,Z 718.765,A -85,B 0,C 180,E1 -17478.27,E2 -17478.27} C_VEL
LIN {X 0,Y 281.24,Z 709.475,A -85,B 0,C 180,E1 -17480.477,E2 -17480.477} C_VEL
LIN {X 0,Y 282.542,Z 698.857,A -85,B 0,C 180,E1 -17482.59,E2 -17482.59} C_VEL
LIN {X 0,Y 283.796,Z 687.398,A -85,B 0,C 180,E1 -17484.506,E2 -17484.506} C_VEL
LIN {X 0,Y 285.248,Z 674.248,A -85,B 0,C 180,E1 -17486.326,E2 -17486.326} C_VEL
LIN {X 0,Y 286.496,Z 660.304,A -85,B 0,C 180,E1 -17487.904,E2 -17487.904} C_VEL
LIN {X 0,Y 287.635,Z 645.331,A -85,B 0,C 180,E1 -17489.253,E2 -17489.253} C_VEL
LIN {X 0,Y 288.526,Z 629.949,A -85,B 0,C 180,E1 -17490.309,E2 -17490.309} C_VEL
LIN {X 0,Y 289.115,Z 614.968,A -85,B 0,C 180,E1 -17491.059,E2 -17491.059} C_VEL
LIN {X 0,Y 289.302,Z 599.206,A -85,B 0,C 180,E1 -17491.65,E2 -17491.65} C_VEL
LIN {X 0,Y 277.297,Z 565.943,A -85,B 0,C 180,E1 -17493.696,E2 -17493.696} C_VEL
LIN {X 0,Y 277.273,Z 565.944,A -85,B 0,C 180,E1 -17497.468,E2 -17497.468} C_VEL
LIN {X 0,Y 277.21,Z 565.951,A -85,B 0,C 180,E1 -17501.235,E2 -17501.235} C_VEL
LIN {X 0,Y 277.201,Z 565.953,A -85,B 0,C 180,E1 -17505.225,E2 -17505.225} C_VEL
LIN {X 0,Y 277.221,Z 565.951,A -85,B 0,C 180,E1 -17508.765,E2 -17508.765} C_VEL
LIN {X 0,Y 277.282,Z 565.947,A -85,B 0,C 180,E1 -17512.532,E2 -17512.532} C_VEL
LIN {X 0,Y 277.254,Z 565.947,A -85,B 0,C 180,E1 -17516.104,E2 -17516.104} C_VEL
LIN {X 0,Y 277.261,Z 565.945,A -85,B 0,C 180,E1 -17519.538,E2 -17519.538} C_VEL
LIN {X 0,Y 277.355,Z 565.937,A -85,B 0,C 180,E1 -17522.863,E2 -17522.863} C_VEL
LIN {X 0,Y 277.327,Z 565.936,A -85,B 0,C 180,E1 -17526.079,E2 -17526.079} C_VEL
LIN {X 0,Y 277.344,Z 565.94,A -85,B 0,C 180,E1 -17530.765,E2 -17530.765} C_VEL
LIN {X 0,Y 277.433,Z 565.924,A -85,B 0,C 180,E1 -17535.325,E2 -17535.325} C_VEL
LIN {X 0,Y 277.505,Z 565.915,A -85,B 0,C 180,E1 -17539.788,E2 -17539.788} C_VEL
LIN {X 0,Y 277.651,Z 565.899,A -85,B 0,C 180,E1 -17542.728,E2 -17542.728} C_VEL
LIN {X 0,Y 277.82,Z 565.877,A -85,B 0,C 180,E1 -17548.55,E2 -17548.55} C_VEL
LIN {X 0,Y 277.82,Z 565.877,A -85,B 0,C 180,E1 -17551.449,E2 -17551.449} C_VEL
LIN {X 0,Y 277.65,Z 565.902,A -85,B 0,C 180,E1 -17557.27,E2 -17557.27} C_VEL
LIN {X 0,Y 277.504,Z 565.914,A -85,B 0,C 180,E1 -17560.21,E2 -17560.21} C_VEL
LIN {X 0,Y 277.432,Z 565.924,A -85,B 0,C 180,E1 -17564.673,E2 -17564.673} C_VEL
LIN {X 0,Y 277.341,Z 565.938,A -85,B 0,C 180,E1 -17569.233,E2 -17569.233} C_VEL
LIN {X 0,Y 277.325,Z 565.94,A -85,B 0,C 180,E1 -17573.92,E2 -17573.92} C_VEL
LIN {X 0,Y 277.322,Z 565.942,A -85,B 0,C 180,E1 -17577.505,E2 -17577.505} C_VEL
LIN {X 0,Y 277.267,Z 565.944,A -85,B 0,C 180,E1 -17580.481,E2 -17580.481} C_VEL
LIN {X 0,Y 277.25,Z 565.951,A -85,B 0,C 180,E1 -17583.894,E2 -17583.894} C_VEL
LIN {X 0,Y 277.284,Z 565.945,A -85,B 0,C 180,E1 -17587.465,E2 -17587.465} C_VEL
LIN {X 0,Y 277.243,Z 565.948,A -85,B 0,C 180,E1 -17591.229,E2 -17591.229} C_VEL
LIN {X 0,Y 277.277,Z 565.944,A -85,B 0,C 180,E1 -17595.209,E2 -17595.209} C_VEL
LIN {X 0,Y 277.34,Z 566.08,A -85,B 0,C 180,E1 -17598.844,E2 -17598.844} C_VEL
LIN {X 0,Y 288.262,Z 595.931,A -85,B 0,C 180,E1 -17600.597,E2 -17600.597} C_VEL
LIN {X 0,Y 287.516,Z 630.485,A -85,B 0,C 180,E1 -17601.784,E2 -17601.784} C_VEL
LIN {X 0,Y 287.013,Z 643.837,A -85,B 0,C 180,E1 -17602.476,E2 -17602.476} C_VEL
LIN {X 0,Y 286.278,Z 657.667,A -85,B 0,C 180,E1 -17603.465,E2 -17603.465} C_VEL
LIN {X 0,Y 285.214,Z 671.31,A -85,B 0,C 180,E1 -17604.745,E2 -17604.745} C_VEL
LIN {X 0,Y 283.926,Z 684.98,A -85,B 0,C 180,E1 -17606.37,E2 -17606.37} C_VEL
LIN {X 0,Y 282.754,Z 695.695,A -85,B 0,C 180,E1 -17607.942,E2 -17607.942} C_VEL
LIN {X 0,Y 281.711,Z 705.424,A -85,B 0,C 180,E1 -17609.657,E2 -17609.657} C_VEL
LIN {X 0,Y 280.609,Z 714.601,A -85,B 0,C 180,E1 -17611.585,E2 -17611.585} C_VEL
LIN {X 0,Y 279.552,Z 723.682,A -85,B 0,C 180,E1 -17613.9,E2 -17613.9} C_VEL
LIN {X 0,Y 278.77,Z 731.112,A -85,B 0,C 180,E1 -17616.212,E2 -17616.212} C_VEL
LIN {X 0,Y 278.124,Z 737.14,A -85,B 0,C 180,E1 -17618.507,E2 -17618.507} C_VEL
LIN {X 0,Y 277.705,Z 741.969,A -85,B 0,C 180,E1 -17620.793,E2 -17620.793} C_VEL
LIN {X 0,Y 277.496,Z 745.733,A -85,B 0,C 180,E1 -17623.068,E2 -17623.068} C_VEL
LIN {X 0,Y 277.517,Z 748.532,A -85,B 0,C 180,E1 -17625.331,E2 -17625.331} C_VEL
LIN {X 0,Y 277.828,Z 750.838,A -85,B 0,C 180,E1 -17628.325,E2 -17628.325} C_VEL
LIN {X 0,Y 278.201,Z 751.537,A -85,B 0,C 180,E1 -17630.134,E2 -17630.134} C_VEL
LIN {X 0,Y 278.91,Z 751.53,A -85,B 0,C 180,E1 -17632.763,E2 -17632.763} C_VEL
LIN {X 0,Y 279.249,Z 751.199,A -85,B 0,C 180,E1 -17633.651,E2 -17633.651} C_VEL
LIN {X 0,Y 279.135,Z 750.783,A -85,B 0,C 180,E1 -17634.861,E2 -17634.861} C_VEL
LIN {X 0,Y 277.344,Z 750.001,A -85,B 0,C 180,E1 -17636.865,E2 -17636.865} C_VEL
LIN {X 0,Y 275.745,Z 748.578,A -85,B 0,C 180,E1 -17638.873,E2 -17638.873} C_VEL
LIN {X 0,Y 275.927,Z 747.156,A -85,B 0,C 180,E1 -17640.065,E2 -17640.065} C_VEL
LIN {X 0,Y 278.292,Z 742.271,A -85,B 0,C 180,E1 -17642.896,E2 -17642.896} C_VEL
LIN {X 0,Y 280.337,Z 737.42,A -85,B 0,C 180,E1 -17645.034,E2 -17645.034} C_VEL
LIN {X 0,Y 282.747,Z 731.393,A -85,B 0,C 180,E1 -17647.14,E2 -17647.14} C_VEL
LIN {X 0,Y 285.648,Z 723.235,A -85,B 0,C 180,E1 -17649.424,E2 -17649.424} C_VEL
LIN {X 0,Y 288.608,Z 713.537,A -85,B 0,C 180,E1 -17651.59,E2 -17651.59} C_VEL
LIN {X 0,Y 291.453,Z 703.286,A -85,B 0,C 180,E1 -17653.421,E2 -17653.421} C_VEL
LIN {X 0,Y 294.075,Z 691.908,A -85,B 0,C 180,E1 -17655.065,E2 -17655.065} C_VEL
LIN {X 0,Y 296.552,Z 679.017,A -85,B 0,C 180,E1 -17656.523,E2 -17656.523} C_VEL
LIN {X 0,Y 298.349,Z 666.628,A -85,B 0,C 180,E1 -17657.656,E2 -17657.656} C_VEL
LIN {X 0,Y 299.659,Z 653.751,A -85,B 0,C 180,E1 -17658.56,E2 -17658.56} C_VEL
LIN {X 0,Y 300.548,Z 638.74,A -85,B 0,C 180,E1 -17659.314,E2 -17659.314} C_VEL
LIN {X 0,Y 302.137,Z 612.84,A -85,B 0,C 180,E1 -17660.314,E2 -17660.314} C_VEL
LIN {X 0,Y 297.377,Z 603.75,A -85,B 0,C 180,E1 -17662.055,E2 -17662.055} C_VEL
LIN {X 0,Y 292.864,Z 596.554,A -85,B 0,C 180,E1 -17663.895,E2 -17663.895} C_VEL
LIN {X 0,Y 290.238,Z 592.65,A -85,B 0,C 180,E1 -17665.092,E2 -17665.092} C_VEL
LIN {X 0,Y 287.509,Z 588.541,A -85,B 0,C 180,E1 -17666.516,E2 -17666.516} C_VEL
LIN {X 0,Y 285.097,Z 585.424,A -85,B 0,C 180,E1 -17667.929,E2 -17667.929} C_VEL
LIN {X 0,Y 284.331,Z 583.995,A -85,B 0,C 180,E1 -17668.465,E2 -17668.465} C_VEL
LIN {X 0,Y 281.712,Z 581.497,A -85,B 0,C 180,E1 -17670.321,E2 -17670.321} C_VEL
LIN {X 0,Y 280.355,Z 578.668,A -85,B 0,C 180,E1 -17671.765,E2 -17671.765} C_VEL
LIN {X 0,Y 277.538,Z 576.685,A -85,B 0,C 180,E1 -17675.622,E2 -17675.622} C_VEL
LIN {X 0,Y 277.054,Z 576.08,A -85,B 0,C 180,E1 -17678.154,E2 -17678.154} C_VEL
LIN {X 0,Y 277.472,Z 576.679,A -85,B 0,C 180,E1 -17680.8,E2 -17680.8} C_VEL
LIN {X 0,Y 280.14,Z 578.581,A -85,B 0,C 180,E1 -17684.625,E2 -17684.625} C_VEL
LIN {X 0,Y 280.592,Z 579.297,A -85,B 0,C 180,E1 -17685.103,E2 -17685.103} C_VEL
LIN {X 0,Y 282.248,Z 582.367,A -85,B 0,C 180,E1 -17686.747,E2 -17686.747} C_VEL
LIN {X 0,Y 283.944,Z 584.039,A -85,B 0,C 180,E1 -17687.949,E2 -17687.949} C_VEL
LIN {X 0,Y 286.897,Z 595.062,A -85,B 0,C 180,E1 -17690.509,E2 -17690.509} C_VEL
LIN {X 0,Y 287.79,Z 597.752,A -85,B 0,C 180,E1 -17691.115,E2 -17691.115} C_VEL
LIN {X 0,Y 289.837,Z 605.544,A -85,B 0,C 180,E1 -17692.53,E2 -17692.53} C_VEL
LIN {X 0,Y 290.522,Z 608.091,A -85,B 0,C 180,E1 -17692.969,E2 -17692.969} C_VEL
LIN {X 0,Y 292.271,Z 623.196,A -85,B 0,C 180,E1 -17694.642,E2 -17694.642} C_VEL
LIN {X 0,Y 293.952,Z 641.208,A -85,B 0,C 180,E1 -17696.319,E2 -17696.319} C_VEL
LIN {X 0,Y 295.139,Z 658.833,A -85,B 0,C 180,E1 -17697.708,E2 -17697.708} C_VEL
LIN {X 0,Y 295.653,Z 691.635,A -85,B 0,C 180,E1 -17699.699,E2 -17699.699} C_VEL
LIN {X 0,Y 293.777,Z 711.515,A -85,B 0,C 180,E1 -17700.51,E2 -17700.51} C_VEL
LIN {X 0,Y 291.548,Z 725.526,A -85,B 0,C 180,E1 -17701.276,E2 -17701.276} C_VEL
LIN {X 0,Y 288.84,Z 739.103,A -85,B 0,C 180,E1 -17702.268,E2 -17702.268} C_VEL
LIN {X 0,Y 285.732,Z 752.489,A -85,B 0,C 180,E1 -17703.526,E2 -17703.526} C_VEL
LIN {X 0,Y 282.281,Z 765.865,A -85,B 0,C 180,E1 -17705.158,E2 -17705.158} C_VEL
LIN {X 0,Y 279.47,Z 775.849,A -85,B 0,C 180,E1 -17706.668,E2 -17706.668} C_VEL
LIN {X 0,Y 276.765,Z 785.305,A -85,B 0,C 180,E1 -17708.396,E2 -17708.396} C_VEL
LIN {X 0,Y 274.166,Z 794.748,A -85,B 0,C 180,E1 -17710.535,E2 -17710.535} C_VEL
LIN {X 0,Y 271.894,Z 803.602,A -85,B 0,C 180,E1 -17713.018,E2 -17713.018} C_VEL
LIN {X 0,Y 270.285,Z 811.116,A -85,B 0,C 180,E1 -17715.7,E2 -17715.7} C_VEL
LIN {X 0,Y 269.26,Z 817.539,A -85,B 0,C 180,E1 -17718.712,E2 -17718.712} C_VEL
LIN {X 0,Y 269.107,Z 821.15,A -85,B 0,C 180,E1 -17720.986,E2 -17720.986} C_VEL
LIN {X 0,Y 269.242,Z 823.263,A -85,B 0,C 180,E1 -17722.711,E2 -17722.711} C_VEL
LIN {X 0,Y 269.8,Z 825.463,A -85,B 0,C 180,E1 -17725.519,E2 -17725.519} C_VEL
LIN {X 0,Y 270.1,Z 826.011,A -85,B 0,C 180,E1 -17727.018,E2 -17727.018} C_VEL
LIN {X 0,Y 270.5,Z 826.137,A -85,B 0,C 180,E1 -17728.512,E2 -17728.512} C_VEL
LIN {X 0,Y 270.72,Z 826.982,A -85,B 0,C 180,E1 -17730.001,E2 -17730.001} C_VEL
LIN {X 0,Y 270.267,Z 827.454,A -85,B 0,C 180,E1 -17731.491,E2 -17731.491} C_VEL
LIN {X 0,Y 269.881,Z 827.489,A -85,B 0,C 180,E1 -17732.986,E2 -17732.986} C_VEL
LIN {X 0,Y 269.638,Z 827.102,A -85,B 0,C 180,E1 -17734.486,E2 -17734.486} C_VEL
LIN {X 0,Y 269.125,Z 825.358,A -85,B 0,C 180,E1 -17737.091,E2 -17737.091} C_VEL
LIN {X 0,Y 268.982,Z 822.27,A -85,B 0,C 180,E1 -17739.779,E2 -17739.779} C_VEL
LIN {X 0,Y 269.305,Z 818.626,A -85,B 0,C 180,E1 -17742.051,E2 -17742.051} C_VEL
LIN {X 0,Y 270.171,Z 814.035,A -85,B 0,C 180,E1 -17744.308,E2 -17744.308} C_VEL
LIN {X 0,Y 271.463,Z 808.039,A -85,B 0,C 180,E1 -17746.681,E2 -17746.681} C_VEL
LIN {X 0,Y 274.194,Z 799.119,A -85,B 0,C 180,E1 -17749.464,E2 -17749.464} C_VEL
LIN {X 0,Y 277.468,Z 789.126,A -85,B 0,C 180,E1 -17751.939,E2 -17751.939} C_VEL
LIN {X 0,Y 280.972,Z 778.815,A -85,B 0,C 180,E1 -17753.984,E2 -17753.984} C_VEL
LIN {X 0,Y 284.938,Z 766.594,A -85,B 0,C 180,E1 -17755.965,E2 -17755.965} C_VEL
LIN {X 0,Y 289.254,Z 753.17,A -85,B 0,C 180,E1 -17757.69,E2 -17757.69} C_VEL
LIN {X 0,Y 293.59,Z 738.344,A -85,B 0,C 180,E1 -17759.193,E2 -17759.193} C_VEL
LIN {X 0,Y 297.564,Z 722.955,A -85,B 0,C 180,E1 -17760.42,E2 -17760.42} C_VEL
LIN {X 0,Y 301.311,Z 705.747,A -85,B 0,C 180,E1 -17761.46,E2 -17761.46} C_VEL
LIN {X 0,Y 303.729,Z 690.096,A -85,B 0,C 180,E1 -17762.236,E2 -17762.236} C_VEL
LIN {X 0,Y 305.464,Z 664.562,A -85,B 0,C 180,E1 -17763.672,E2 -17763.672} C_VEL
LIN {X 0,Y 305.942,Z 649.453,A -85,B 0,C 180,E1 -17764.76,E2 -17764.76} C_VEL
LIN {X 0,Y 305.948,Z 634.374,A -85,B 0,C 180,E1 -17766.144,E2 -17766.144} C_VEL
LIN {X 0,Y 305.723,Z 621.301,A -85,B 0,C 180,E1 -17767.595,E2 -17767.595} C_VEL
LIN {X 0,Y 305.571,Z 611.62,A -85,B 0,C 180,E1 -17768.853,E2 -17768.853} C_VEL
LIN {X 0,Y 305.105,Z 608.579,A -85,B 0,C 180,E1 -17769.55,E2 -17769.55} C_VEL
LIN {X 0,Y 304.304,Z 606.984,A -85,B 0,C 180,E1 -17770.345,E2 -17770.345} C_VEL
LIN {X 0,Y 302.511,Z 603.921,A -85,B 0,C 180,E1 -17772.72,E2 -17772.72} C_VEL
LIN {X 0,Y 302.208,Z 602.763,A -85,B 0,C 180,E1 -17773.593,E2 -17773.593} C_VEL
LIN {X 0,Y 301.722,Z 602.532,A -85,B 0,C 180,E1 -17776.227,E2 -17776.227} C_VEL
LIN {X 0,Y 302.555,Z 602.976,A -85,B 0,C 180,E1 -17778.505,E2 -17778.505} C_VEL
LIN {X 0,Y 303.808,Z 606.074,A -85,B 0,C 180,E1 -17780.517,E2 -17780.517} C_VEL
LIN {X 0,Y 305.128,Z 607.635,A -85,B 0,C 180,E1 -17781.694,E2 -17781.694} C_VEL
LIN {X 0,Y 307.405,Z 611.731,A -85,B 0,C 180,E1 -17783.442,E2 -17783.442} C_VEL
LIN {X 0,Y 309.953,Z 616.44,A -85,B 0,C 180,E1 -17784.994,E2 -17784.994} C_VEL
LIN {X 0,Y 312.144,Z 620.881,A -85,B 0,C 180,E1 -17786.129,E2 -17786.129} C_VEL
LIN {X 0,Y 310.399,Z 643.8,A -85,B 0,C 180,E1 -17787.228,E2 -17787.228} C_VEL
LIN {X 0,Y 308.715,Z 658.207,A -85,B 0,C 180,E1 -17788.163,E2 -17788.163} C_VEL
LIN {X 0,Y 306.315,Z 672.864,A -85,B 0,C 180,E1 -17789.408,E2 -17789.408} C_VEL
LIN {X 0,Y 303.97,Z 683.979,A -85,B 0,C 180,E1 -17790.572,E2 -17790.572} C_VEL
LIN {X 0,Y 301.13,Z 695.046,A -85,B 0,C 180,E1 -17791.985,E2 -17791.985} C_VEL
LIN {X 0,Y 297.97,Z 705.743,A -85,B 0,C 180,E1 -17793.624,E2 -17793.624} C_VEL
LIN {X 0,Y 294.463,Z 715.992,A -85,B 0,C 180,E1 -17795.554,E2 -17795.554} C_VEL
LIN {X 0,Y 290.418,Z 726.369,A -85,B 0,C 180,E1 -17797.969,E2 -17797.969} C_VEL
LIN {X 0,Y 286.899,Z 734.364,A -85,B 0,C 180,E1 -17800.316,E2 -17800.316} C_VEL
LIN {X 0,Y 283.719,Z 740.844,A -85,B 0,C 180,E1 -17802.707,E2 -17802.707} C_VEL
LIN {X 0,Y 280.498,Z 746.72,A -85,B 0,C 180,E1 -17805.489,E2 -17805.489} C_VEL
LIN {X 0,Y 277.696,Z 751.052,A -85,B 0,C 180,E1 -17808.318,E2 -17808.318} C_VEL
LIN {X 0,Y 275.575,Z 753.997,A -85,B 0,C 180,E1 -17811.197,E2 -17811.197} C_VEL
LIN {X 0,Y 273.774,Z 755.683,A -85,B 0,C 180,E1 -17814.106,E2 -17814.106} C_VEL
LIN {X 0,Y 272.412,Z 756.114,A -85,B 0,C 180,E1 -17817.042,E2 -17817.042} C_VEL
LIN {X 0,Y 271.485,Z 755.301,A -85,B 0,C 180,E1 -17819.999,E2 -17819.999} C_VEL
LIN {X 0,Y 270.882,Z 753.237,A -85,B 0,C 180,E1 -17822.974,E2 -17822.974} C_VEL
LIN {X 0,Y 270.599,Z 749.881,A -85,B 0,C 180,E1 -17825.962,E2 -17825.962} C_VEL
LIN {X 0,Y 270.762,Z 746.46,A -85,B 0,C 180,E1 -17828.207,E2 -17828.207} C_VEL
LIN {X 0,Y 271.044,Z 740.642,A -85,B 0,C 180,E1 -17831.213,E2 -17831.213} C_VEL
LIN {X 0,Y 271.551,Z 734.166,A -85,B 0,C 180,E1 -17833.85,E2 -17833.85} C_VEL
LIN {X 0,Y 272.405,Z 726.246,A -85,B 0,C 180,E1 -17836.486,E2 -17836.486} C_VEL
LIN {X 0,Y 273.508,Z 716.61,A -85,B 0,C 180,E1 -17839.124,E2 -17839.124} C_VEL
LIN {X 0,Y 274.678,Z 706.669,A -85,B 0,C 180,E1 -17841.383,E2 -17841.383} C_VEL
LIN {X 0,Y 276.125,Z 694.421,A -85,B 0,C 180,E1 -17843.687,E2 -17843.687} C_VEL
LIN {X 0,Y 277.58,Z 681.484,A -85,B 0,C 180,E1 -17845.695,E2 -17845.695} C_VEL
LIN {X 0,Y 278.9,Z 668.299,A -85,B 0,C 180,E1 -17847.379,E2 -17847.379} C_VEL
LIN {X 0,Y 280.148,Z 653.852,A -85,B 0,C 180,E1 -17848.875,E2 -17848.875} C_VEL
LIN {X 0,Y 281.194,Z 638.895,A -85,B 0,C 180,E1 -17850.092,E2 -17850.092} C_VEL
LIN {X 0,Y 281.979,Z 623.551,A -85,B 0,C 180,E1 -17851.027,E2 -17851.027} C_VEL
LIN {X 0,Y 282.453,Z 605.59,A -85,B 0,C 180,E1 -17851.795,E2 -17851.795} C_VEL
LIN {X 0,Y 282.474,Z 600.892,A -85,B 0,C 180,E1 -17851.976,E2 -17851.976} C_VEL
LIN {X 0,Y 270.24,Z 566.986,A -85,B 0,C 180,E1 -17854.087,E2 -17854.087} C_VEL
LIN {X 0,Y 270.229,Z 566.822,A -85,B 0,C 180,E1 -17856.738,E2 -17856.738} C_VEL
LIN {X 0,Y 270.17,Z 566.828,A -85,B 0,C 180,E1 -17861.027,E2 -17861.027} C_VEL
LIN {X 0,Y 270.153,Z 566.831,A -85,B 0,C 180,E1 -17865.379,E2 -17865.379} C_VEL
LIN {X 0,Y 270.183,Z 566.825,A -85,B 0,C 180,E1 -17869.435,E2 -17869.435} C_VEL
LIN {X 0,Y 270.255,Z 566.818,A -85,B 0,C 180,E1 -17873.721,E2 -17873.721} C_VEL
LIN {X 0,Y 270.203,Z 566.825,A -85,B 0,C 180,E1 -17876.892,E2 -17876.892} C_VEL
LIN {X 0,Y 270.194,Z 566.828,A -85,B 0,C 180,E1 -17880.382,E2 -17880.382} C_VEL
LIN {X 0,Y 270.261,Z 566.817,A -85,B 0,C 180,E1 -17883.763,E2 -17883.763} C_VEL
LIN {X 0,Y 270.232,Z 566.822,A -85,B 0,C 180,E1 -17887.038,E2 -17887.038} C_VEL
LIN {X 0,Y 270.301,Z 566.813,A -85,B 0,C 180,E1 -17890.244,E2 -17890.244} C_VEL
LIN {X 0,Y 270.402,Z 566.802,A -85,B 0,C 180,E1 -17894.934,E2 -17894.934} C_VEL
LIN {X 0,Y 270.44,Z 566.796,A -85,B 0,C 180,E1 -17899.518,E2 -17899.518} C_VEL
LIN {X 0,Y 270.61,Z 566.775,A -85,B 0,C 180,E1 -17902.538,E2 -17902.538} C_VEL
LIN {X 0,Y 270.786,Z 566.753,A -85,B 0,C 180,E1 -17908.512,E2 -17908.512} C_VEL
LIN {X 0,Y 270.785,Z 566.753,A -85,B 0,C 180,E1 -17911.486,E2 -17911.486} C_VEL
LIN {X 0,Y 270.608,Z 566.778,A -85,B 0,C 180,E1 -17917.46,E2 -17917.46} C_VEL
LIN {X 0,Y 270.439,Z 566.794,A -85,B 0,C 180,E1 -17920.48,E2 -17920.48} C_VEL
LIN {X 0,Y 270.4,Z 566.802,A -85,B 0,C 180,E1 -17925.064,E2 -17925.064} C_VEL
LIN {X 0,Y 270.298,Z 566.814,A -85,B 0,C 180,E1 -17929.755,E2 -17929.755} C_VEL
LIN {X 0,Y 270.27,Z 566.816,A -85,B 0,C 180,E1 -17934.585,E2 -17934.585} C_VEL
LIN {X 0,Y 270.266,Z 566.818,A -85,B 0,C 180,E1 -17937.908,E2 -17937.908} C_VEL
LIN {X 0,Y 270.18,Z 566.828,A -85,B 0,C 180,E1 -17941.348,E2 -17941.348} C_VEL
LIN {X 0,Y 270.211,Z 566.823,A -85,B 0,C 180,E1 -17944.903,E2 -17944.903} C_VEL
LIN {X 0,Y 270.217,Z 566.823,A -85,B 0,C 180,E1 -17948.717,E2 -17948.717} C_VEL
LIN {X 0,Y 270.209,Z 566.825,A -85,B 0,C 180,E1 -17952.55,E2 -17952.55} C_VEL
LIN {X 0,Y 270.225,Z 566.823,A -85,B 0,C 180,E1 -17956.736,E2 -17956.736} C_VEL
LIN {X 0,Y 270.257,Z 566.891,A -85,B 0,C 180,E1 -17958.385,E2 -17958.385} C_VEL
LIN {X 0,Y 281.495,Z 597.634,A -85,B 0,C 180,E1 -17960.253,E2 -17960.253} C_VEL
LIN {X 0,Y 280.639,Z 631.885,A -85,B 0,C 180,E1 -17961.47,E2 -17961.47} C_VEL
LIN {X 0,Y 280.037,Z 646.81,A -85,B 0,C 180,E1 -17962.286,E2 -17962.286} C_VEL
LIN {X 0,Y 279.151,Z 661.213,A -85,B 0,C 180,E1 -17963.395,E2 -17963.395} C_VEL
LIN {X 0,Y 278.12,Z 674.2,A -85,B 0,C 180,E1 -17964.688,E2 -17964.688} C_VEL
LIN {X 0,Y 276.883,Z 686.551,A -85,B 0,C 180,E1 -17966.219,E2 -17966.219} C_VEL
LIN {X 0,Y 275.58,Z 698.448,A -85,B 0,C 180,E1 -17968.051,E2 -17968.051} C_VEL
LIN {X 0,Y 274.364,Z 709.036,A -85,B 0,C 180,E1 -17970.034,E2 -17970.034} C_VEL
LIN {X 0,Y 273.133,Z 719.443,A -85,B 0,C 180,E1 -17972.41,E2 -17972.41} C_VEL
LIN {X 0,Y 272.221,Z 727.382,A -85,B 0,C 180,E1 -17974.633,E2 -17974.633} C_VEL
LIN {X 0,Y 271.382,Z 734.71,A -85,B 0,C 180,E1 -17977.142,E2 -17977.142} C_VEL
LIN {X 0,Y 270.852,Z 740.569,A -85,B 0,C 180,E1 -17979.649,E2 -17979.649} C_VEL
LIN {X 0,Y 270.495,Z 745.911,A -85,B 0,C 180,E1 -17982.616,E2 -17982.616} C_VEL
LIN {X 0,Y 270.47,Z 748.957,A -85,B 0,C 180,E1 -17984.94,E2 -17984.94} C_VEL
LIN {X 0,Y 270.581,Z 750.506,A -85,B 0,C 180,E1 -17986.482,E2 -17986.482} C_VEL
LIN {X 0,Y 270.75,Z 751.654,A -85,B 0,C 180,E1 -17988.015,E2 -17988.015} C_VEL
LIN {X 0,Y 271.395,Z 752.77,A -85,B 0,C 180,E1 -17991.062,E2 -17991.062} C_VEL
LIN {X 0,Y 272.452,Z 752.421,A -85,B 0,C 180,E1 -17994.078,E2 -17994.078} C_VEL
LIN {X 0,Y 273.965,Z 750.617,A -85,B 0,C 180,E1 -17997.06,E2 -17997.06} C_VEL
LIN {X 0,Y 275.879,Z 747.249,A -85,B 0,C 180,E1 -18000.001,E2 -18000.001} C_VEL
LIN {X 0,Y 275.927,Z 747.156,A -85,B 0,C 180,E1 -18000.065,E2 -18000.065} C_VEL
LIN {X 0,Y 276.196,Z 745.571,A -85,B 0,C 180,E1 -18001.246,E2 -18001.246} C_VEL
LIN {X 0,Y 275.112,Z 743.015,A -85,B 0,C 180,E1 -18003.228,E2 -18003.228} C_VEL
LIN {X 0,Y 274.228,Z 739.895,A -85,B 0,C 180,E1 -18005.18,E2 -18005.18} C_VEL
LIN {X 0,Y 274.784,Z 737.397,A -85,B 0,C 180,E1 -18006.289,E2 -18006.289} C_VEL
LIN {X 0,Y 277.81,Z 730.087,A -85,B 0,C 180,E1 -18008.731,E2 -18008.731} C_VEL
LIN {X 0,Y 280.716,Z 722.257,A -85,B 0,C 180,E1 -18010.823,E2 -18010.823} C_VEL
LIN {X 0,Y 283.742,Z 712.784,A -85,B 0,C 180,E1 -18012.881,E2 -18012.881} C_VEL
LIN {X 0,Y 287.098,Z 700.906,A -85,B 0,C 180,E1 -18014.895,E2 -18014.895} C_VEL
LIN {X 0,Y 289.653,Z 690.107,A -85,B 0,C 180,E1 -18016.384,E2 -18016.384} C_VEL
LIN {X 0,Y 291.967,Z 678.243,A -85,B 0,C 180,E1 -18017.693,E2 -18017.693} C_VEL
LIN {X 0,Y 293.819,Z 665.106,A -85,B 0,C 180,E1 -18018.84,E2 -18018.84} C_VEL
LIN {X 0,Y 295.25,Z 651.255,A -85,B 0,C 180,E1 -18019.765,E2 -18019.765} C_VEL
LIN {X 0,Y 296.397,Z 631.694,A -85,B 0,C 180,E1 -18020.665,E2 -18020.665} C_VEL
LIN {X 0,Y 297.493,Z 616.048,A -85,B 0,C 180,E1 -18021.284,E2 -18021.284} C_VEL
LIN {X 0,Y 293.441,Z 608.147,A -85,B 0,C 180,E1 -18022.907,E2 -18022.907} C_VEL
LIN {X 0,Y 289.478,Z 601.722,A -85,B 0,C 180,E1 -18024.655,E2 -18024.655} C_VEL
LIN {X 0,Y 287.349,Z 598.409,A -85,B 0,C 180,E1 -18025.724,E2 -18025.724} C_VEL
LIN {X 0,Y 285.091,Z 594.88,A -85,B 0,C 180,E1 -18026.982,E2 -18026.982} C_VEL
LIN {X 0,Y 282.615,Z 591.35,A -85,B 0,C 180,E1 -18028.551,E2 -18028.551} C_VEL
LIN {X 0,Y 281.93,Z 590.349,A -85,B 0,C 180,E1 -18029.052,E2 -18029.052} C_VEL
LIN {X 0,Y 279.672,Z 587.854,A -85,B 0,C 180,E1 -18030.819,E2 -18030.819} C_VEL
LIN {X 0,Y 278.653,Z 585.562,A -85,B 0,C 180,E1 -18031.982,E2 -18031.982} C_VEL
LIN {X 0,Y 276.025,Z 583.557,A -85,B 0,C 180,E1 -18035.847,E2 -18035.847} C_VEL
LIN {X 0,Y 275.637,Z 583.051,A -85,B 0,C 180,E1 -18037.777,E2 -18037.777} C_VEL
LIN {X 0,Y 275.909,Z 583.478,A -85,B 0,C 180,E1 -18040.352,E2 -18040.352} C_VEL
LIN {X 0,Y 278.188,Z 585.3,A -85,B 0,C 180,E1 -18044.117,E2 -18044.117} C_VEL
LIN {X 0,Y 278.609,Z 585.635,A -85,B 0,C 180,E1 -18044.588,E2 -18044.588} C_VEL
LIN {X 0,Y 280.275,Z 588.935,A -85,B 0,C 180,E1 -18046.386,E2 -18046.386} C_VEL
LIN {X 0,Y 281.608,Z 590.466,A -85,B 0,C 180,E1 -18047.411,E2 -18047.411} C_VEL
LIN {X 0,Y 284.079,Z 600.566,A -85,B 0,C 180,E1 -18049.821,E2 -18049.821} C_VEL
LIN {X 0,Y 284.749,Z 603.183,A -85,B 0,C 180,E1 -18050.377,E2 -18050.377} C_VEL
LIN {X 0,Y 286.922,Z 612.208,A -85,B 0,C 180,E1 -18052.06,E2 -18052.06} C_VEL
LIN {X 0,Y 288.294,Z 627.069,A -85,B 0,C 180,E1 -18053.728,E2 -18053.728} C_VEL
LIN {X 0,Y 289.663,Z 644.115,A -85,B 0,C 180,E1 -18055.367,E2 -18055.367} C_VEL
LIN {X 0,Y 290.543,Z 661.259,A -85,B 0,C 180,E1 -18056.741,E2 -18056.741} C_VEL
LIN {X 0,Y 290.744,Z 692.64,A -85,B 0,C 180,E1 -18058.713,E2 -18058.713} C_VEL
LIN {X 0,Y 288.851,Z 710.543,A -85,B 0,C 180,E1 -18059.477,E2 -18059.477} C_VEL
LIN {X 0,Y 286.137,Z 726.2,A -85,B 0,C 180,E1 -18060.377,E2 -18060.377} C_VEL
LIN {X 0,Y 283.099,Z 740.214,A -85,B 0,C 180,E1 -18061.454,E2 -18061.454} C_VEL
LIN {X 0,Y 279.504,Z 754.361,A -85,B 0,C 180,E1 -18062.888,E2 -18062.888} C_VEL
LIN {X 0,Y 275.928,Z 767.024,A -85,B 0,C 180,E1 -18064.545,E2 -18064.545} C_VEL
LIN {X 0,Y 273.002,Z 776.608,A -85,B 0,C 180,E1 -18066.081,E2 -18066.081} C_VEL
LIN {X 0,Y 269.741,Z 787.304,A -85,B 0,C 180,E1 -18068.207,E2 -18068.207} C_VEL
LIN {X 0,Y 267.075,Z 796.22,A -85,B 0,C 180,E1 -18070.397,E2 -18070.397} C_VEL
LIN {X 0,Y 264.687,Z 804.688,A -85,B 0,C 180,E1 -18073.019,E2 -18073.019} C_VEL
LIN {X 0,Y 263.336,Z 810.643,A -85,B 0,C 180,E1 -18075.314,E2 -18075.314} C_VEL
LIN {X 0,Y 262.406,Z 815.474,A -85,B 0,C 180,E1 -18077.629,E2 -18077.629} C_VEL
LIN {X 0,Y 262.037,Z 820.35,A -85,B 0,C 180,E1 -18080.74,E2 -18080.74} C_VEL
LIN {X 0,Y 262.17,Z 822.501,A -85,B 0,C 180,E1 -18082.689,E2 -18082.689} C_VEL
LIN {X 0,Y 262.728,Z 824.416,A -85,B 0,C 180,E1 -18085.398,E2 -18085.398} C_VEL
LIN {X 0,Y 263.046,Z 824.912,A -85,B 0,C 180,E1 -18086.938,E2 -18086.938} C_VEL
LIN {X 0,Y 263.47,Z 824.973,A -85,B 0,C 180,E1 -18088.472,E2 -18088.472} C_VEL
LIN {X 0,Y 263.753,Z 825.638,A -85,B 0,C 180,E1 -18090.001,E2 -18090.001} C_VEL
LIN {X 0,Y 263.257,Z 826.179,A -85,B 0,C 180,E1 -18091.531,E2 -18091.531} C_VEL
LIN {X 0,Y 262.853,Z 826.286,A -85,B 0,C 180,E1 -18093.066,E2 -18093.066} C_VEL
LIN {X 0,Y 262.574,Z 825.968,A -85,B 0,C 180,E1 -18094.607,E2 -18094.607} C_VEL
LIN {X 0,Y 262.004,Z 824.026,A -85,B 0,C 180,E1 -18097.709,E2 -18097.709} C_VEL
LIN {X 0,Y 261.975,Z 820.449,A -85,B 0,C 180,E1 -18100.825,E2 -18100.825} C_VEL
LIN {X 0,Y 262.604,Z 816.667,A -85,B 0,C 180,E1 -18103.15,E2 -18103.15} C_VEL
LIN {X 0,Y 263.652,Z 811.935,A -85,B 0,C 180,E1 -18105.461,E2 -18105.461} C_VEL
LIN {X 0,Y 265.217,Z 806.194,A -85,B 0,C 180,E1 -18107.743,E2 -18107.743} C_VEL
LIN {X 0,Y 267.933,Z 798.068,A -85,B 0,C 180,E1 -18110.339,E2 -18110.339} C_VEL
LIN {X 0,Y 271.588,Z 788.218,A -85,B 0,C 180,E1 -18112.841,E2 -18112.841} C_VEL
LIN {X 0,Y 275.203,Z 778.156,A -85,B 0,C 180,E1 -18114.922,E2 -18114.922} C_VEL
LIN {X 0,Y 279.432,Z 766.2,A -85,B 0,C 180,E1 -18116.919,E2 -18116.919} C_VEL
LIN {X 0,Y 284.406,Z 751.851,A -85,B 0,C 180,E1 -18118.808,E2 -18118.808} C_VEL
LIN {X 0,Y 288.977,Z 737.302,A -85,B 0,C 180,E1 -18120.309,E2 -18120.309} C_VEL
LIN {X 0,Y 293.43,Z 721.355,A -85,B 0,C 180,E1 -18121.597,E2 -18121.597} C_VEL
LIN {X 0,Y 297.616,Z 703.265,A -85,B 0,C 180,E1 -18122.696,E2 -18122.696} C_VEL
LIN {X 0,Y 299.667,Z 690.986,A -85,B 0,C 180,E1 -18123.338,E2 -18123.338} C_VEL
LIN {X 0,Y 301.794,Z 666.283,A -85,B 0,C 180,E1 -18124.768,E2 -18124.768} C_VEL
LIN {X 0,Y 302.497,Z 651.563,A -85,B 0,C 180,E1 -18125.863,E2 -18125.863} C_VEL
LIN {X 0,Y 302.806,Z 637.361,A -85,B 0,C 180,E1 -18127.198,E2 -18127.198} C_VEL
LIN {X 0,Y 302.944,Z 625.119,A -85,B 0,C 180,E1 -18128.588,E2 -18128.588} C_VEL
LIN {X 0,Y 303.045,Z 616.148,A -85,B 0,C 180,E1 -18129.785,E2 -18129.785} C_VEL
LIN {X 0,Y 302.807,Z 614.464,A -85,B 0,C 180,E1 -18130.21,E2 -18130.21} C_VEL
LIN {X 0,Y 302.35,Z 613.582,A -85,B 0,C 180,E1 -18130.724,E2 -18130.724} C_VEL
LIN {X 0,Y 300.826,Z 610.581,A -85,B 0,C 180,E1 -18133.044,E2 -18133.044} C_VEL
LIN {X 0,Y 300.689,Z 609.805,A -85,B 0,C 180,E1 -18133.567,E2 -18133.567} C_VEL
LIN {X 0,Y 300.277,Z 609.505,A -85,B 0,C 180,E1 -18136.516,E2 -18136.516} C_VEL
LIN {X 0,Y 300.928,Z 609.828,A -85,B 0,C 180,E1 -18138.255,E2 -18138.255} C_VEL
LIN {X 0,Y 302.294,Z 613.071,A -85,B 0,C 180,E1 -18140.493,E2 -18140.493} C_VEL
LIN {X 0,Y 303.279,Z 614.514,A -85,B 0,C 180,E1 -18141.458,E2 -18141.458} C_VEL
LIN {X 0,Y 305.222,Z 618.153,A -85,B 0,C 180,E1 -18143.037,E2 -18143.037} C_VEL
LIN {X 0,Y 307.909,Z 623.479,A -85,B 0,C 180,E1 -18144.78,E2 -18144.78} C_VEL
LIN {X 0,Y 308.505,Z 625.149,A -85,B 0,C 180,E1 -18145.146,E2 -18145.146} C_VEL
LIN {X 0,Y 306.663,Z 645.937,A -85,B 0,C 180,E1 -18146.17,E2 -18146.17} C_VEL
LIN {X 0,Y 304.56,Z 661.8,A -85,B 0,C 180,E1 -18147.24,E2 -18147.24} C_VEL
LIN {X 0,Y 302.09,Z 675.344,A -85,B 0,C 180,E1 -18148.435,E2 -18148.435} C_VEL
LIN {X 0,Y 299.358,Z 686.828,A -85,B 0,C 180,E1 -18149.684,E2 -18149.684} C_VEL
LIN {X 0,Y 296.384,Z 697.694,A -85,B 0,C 180,E1 -18151.109,E2 -18151.109} C_VEL
LIN {X 0,Y 292.781,Z 708.694,A -85,B 0,C 180,E1 -18152.865,E2 -18152.865} C_VEL
LIN {X 0,Y 289.059,Z 718.701,A -85,B 0,C 180,E1 -18154.817,E2 -18154.817} C_VEL
LIN {X 0,Y 285.569,Z 727.051,A -85,B 0,C 180,E1 -18156.81,E2 -18156.81} C_VEL
LIN {X 0,Y 281.735,Z 735.14,A -85,B 0,C 180,E1 -18159.177,E2 -18159.177} C_VEL
LIN {X 0,Y 278.272,Z 741.74,A -85,B 0,C 180,E1 -18161.596,E2 -18161.596} C_VEL
LIN {X 0,Y 274.772,Z 747.656,A -85,B 0,C 180,E1 -18164.42,E2 -18164.42} C_VEL
LIN {X 0,Y 272.437,Z 751.127,A -85,B 0,C 180,E1 -18166.574,E2 -18166.574} C_VEL
LIN {X 0,Y 269.754,Z 754.523,A -85,B 0,C 180,E1 -18169.491,E2 -18169.491} C_VEL
LIN {X 0,Y 267.766,Z 756.551,A -85,B 0,C 180,E1 -18172.458,E2 -18172.458} C_VEL
LIN {X 0,Y 266.081,Z 757.395,A -85,B 0,C 180,E1 -18175.455,E2 -18175.455} C_VEL
LIN {X 0,Y 264.882,Z 756.971,A -85,B 0,C 180,E1 -18178.479,E2 -18178.479} C_VEL
LIN {X 0,Y 264.128,Z 755.297,A -85,B 0,C 180,E1 -18181.524,E2 -18181.524} C_VEL
LIN {X 0,Y 263.582,Z 752.377,A -85,B 0,C 180,E1 -18184.587,E2 -18184.587} C_VEL
LIN {X 0,Y 263.72,Z 748.086,A -85,B 0,C 180,E1 -18187.657,E2 -18187.657} C_VEL
LIN {X 0,Y 263.934,Z 742.366,A -85,B 0,C 180,E1 -18190.742,E2 -18190.742} C_VEL
LIN {X 0,Y 264.469,Z 735.029,A -85,B 0,C 180,E1 -18193.837,E2 -18193.837} C_VEL
LIN {X 0,Y 265.362,Z 727.05,A -85,B 0,C 180,E1 -18196.541,E2 -18196.541} C_VEL
LIN {X 0,Y 266.461,Z 717.323,A -85,B 0,C 180,E1 -18199.249,E2 -18199.249} C_VEL
LIN {X 0,Y 267.644,Z 707.274,A -85,B 0,C 180,E1 -18201.568,E2 -18201.568} C_VEL
LIN {X 0,Y 269.025,Z 695.958,A -85,B 0,C 180,E1 -18203.748,E2 -18203.748} C_VEL
LIN {X 0,Y 270.485,Z 683.135,A -85,B 0,C 180,E1 -18205.798,E2 -18205.798} C_VEL
LIN {X 0,Y 271.844,Z 670.045,A -85,B 0,C 180,E1 -18207.523,E2 -18207.523} C_VEL
LIN {X 0,Y 273.143,Z 655.418,A -85,B 0,C 180,E1 -18209.088,E2 -18209.088} C_VEL
LIN {X 0,Y 274.185,Z 640.984,A -85,B 0,C 180,E1 -18210.306,E2 -18210.306} C_VEL
LIN {X 0,Y 275.069,Z 625.094,A -85,B 0,C 180,E1 -18211.311,E2 -18211.311} C_VEL
LIN {X 0,Y 275.562,Z 607.016,A -85,B 0,C 180,E1 -18212.11,E2 -18212.11} C_VEL
LIN {X 0,Y 275.475,Z 602.113,A -85,B 0,C 180,E1 -18212.31,E2 -18212.31} C_VEL
LIN {X 0,Y 263.177,Z 567.701,A -85,B 0,C 180,E1 -18214.562,E2 -18214.562} C_VEL
LIN {X 0,Y 263.163,Z 567.704,A -85,B 0,C 180,E1 -18217.895,E2 -18217.895} C_VEL
LIN {X 0,Y 263.124,Z 567.707,A -85,B 0,C 180,E1 -18221.892,E2 -18221.892} C_VEL
LIN {X 0,Y 263.125,Z 567.709,A -85,B 0,C 180,E1 -18226.149,E2 -18226.149} C_VEL
LIN {X 0,Y 263.121,Z 567.708,A -85,B 0,C 180,E1 -18230.129,E2 -18230.129} C_VEL
LIN {X 0,Y 263.188,Z 567.7,A -85,B 0,C 180,E1 -18234.021,E2 -18234.021} C_VEL
LIN {X 0,Y 263.133,Z 567.703,A -85,B 0,C 180,E1 -18237.711,E2 -18237.711} C_VEL
LIN {X 0,Y 263.195,Z 567.698,A -85,B 0,C 180,E1 -18241.784,E2 -18241.784} C_VEL
LIN {X 0,Y 263.225,Z 567.693,A -85,B 0,C 180,E1 -18245.199,E2 -18245.199} C_VEL
LIN {X 0,Y 263.263,Z 567.689,A -85,B 0,C 180,E1 -18249.692,E2 -18249.692} C_VEL
LIN {X 0,Y 263.35,Z 567.68,A -85,B 0,C 180,E1 -18254.521,E2 -18254.521} C_VEL
LIN {X 0,Y 263.373,Z 567.678,A -85,B 0,C 180,E1 -18259.233,E2 -18259.233} C_VEL
LIN {X 0,Y 263.571,Z 567.651,A -85,B 0,C 180,E1 -18262.337,E2 -18262.337} C_VEL
LIN {X 0,Y 263.75,Z 567.629,A -85,B 0,C 180,E1 -18268.472,E2 -18268.472} C_VEL
LIN {X 0,Y 263.75,Z 567.629,A -85,B 0,C 180,E1 -18271.526,E2 -18271.526} C_VEL
LIN {X 0,Y 263.569,Z 567.653,A -85,B 0,C 180,E1 -18277.661,E2 -18277.661} C_VEL
LIN {X 0,Y 263.372,Z 567.676,A -85,B 0,C 180,E1 -18280.765,E2 -18280.765} C_VEL
LIN {X 0,Y 263.348,Z 567.683,A -85,B 0,C 180,E1 -18285.477,E2 -18285.477} C_VEL
LIN {X 0,Y 263.264,Z 567.687,A -85,B 0,C 180,E1 -18290.305,E2 -18290.305} C_VEL
LIN {X 0,Y 263.205,Z 567.699,A -85,B 0,C 180,E1 -18295.291,E2 -18295.291} C_VEL
LIN {X 0,Y 263.172,Z 567.699,A -85,B 0,C 180,E1 -18298.729,E2 -18298.729} C_VEL
LIN {X 0,Y 263.13,Z 567.706,A -85,B 0,C 180,E1 -18302.287,E2 -18302.287} C_VEL
LIN {X 0,Y 263.186,Z 567.702,A -85,B 0,C 180,E1 -18305.977,E2 -18305.977} C_VEL
LIN {X 0,Y 263.152,Z 567.708,A -85,B 0,C 180,E1 -18309.863,E2 -18309.863} C_VEL
LIN {X 0,Y 263.182,Z 567.704,A -85,B 0,C 180,E1 -18313.97,E2 -18313.97} C_VEL
LIN {X 0,Y 263.224,Z 567.821,A -85,B 0,C 180,E1 -18317.929,E2 -18317.929} C_VEL
LIN {X 0,Y 274.65,Z 599.386,A -85,B 0,C 180,E1 -18319.896,E2 -18319.896} C_VEL
LIN {X 0,Y 273.788,Z 632.833,A -85,B 0,C 180,E1 -18321.121,E2 -18321.121} C_VEL
LIN {X 0,Y 273.202,Z 646.557,A -85,B 0,C 180,E1 -18321.875,E2 -18321.875} C_VEL
LIN {X 0,Y 272.473,Z 659.297,A -85,B 0,C 180,E1 -18322.832,E2 -18322.832} C_VEL
LIN {X 0,Y 271.411,Z 672.701,A -85,B 0,C 180,E1 -18324.137,E2 -18324.137} C_VEL
LIN {X 0,Y 270.056,Z 686.246,A -85,B 0,C 180,E1 -18325.805,E2 -18325.805} C_VEL
LIN {X 0,Y 268.752,Z 697.871,A -85,B 0,C 180,E1 -18327.583,E2 -18327.583} C_VEL
LIN {X 0,Y 267.482,Z 708.71,A -85,B 0,C 180,E1 -18329.617,E2 -18329.617} C_VEL
LIN {X 0,Y 266.201,Z 719.351,A -85,B 0,C 180,E1 -18332.056,E2 -18332.056} C_VEL
LIN {X 0,Y 265.222,Z 727.797,A -85,B 0,C 180,E1 -18334.423,E2 -18334.423} C_VEL
LIN {X 0,Y 264.371,Z 735.052,A -85,B 0,C 180,E1 -18336.915,E2 -18336.915} C_VEL
LIN {X 0,Y 263.779,Z 741.577,A -85,B 0,C 180,E1 -18339.736,E2 -18339.736} C_VEL
LIN {X 0,Y 263.465,Z 745.955,A -85,B 0,C 180,E1 -18342.136,E2 -18342.136} C_VEL
LIN {X 0,Y 263.421,Z 749.322,A -85,B 0,C 180,E1 -18344.527,E2 -18344.527} C_VEL
LIN {X 0,Y 263.66,Z 752.34,A -85,B 0,C 180,E1 -18347.688,E2 -18347.688} C_VEL
LIN {X 0,Y 264.329,Z 753.845,A -85,B 0,C 180,E1 -18350.821,E2 -18350.821} C_VEL
LIN {X 0,Y 265.404,Z 753.821,A -85,B 0,C 180,E1 -18353.92,E2 -18353.92} C_VEL
LIN {X 0,Y 266.92,Z 752.322,A -85,B 0,C 180,E1 -18356.982,E2 -18356.982} C_VEL
LIN {X 0,Y 268.92,Z 749.347,A -85,B 0,C 180,E1 -18360.001,E2 -18360.001} C_VEL
LIN {X 0,Y 270.75,Z 746.061,A -85,B 0,C 180,E1 -18362.232,E2 -18362.232} C_VEL
LIN {X 0,Y 272.822,Z 741.839,A -85,B 0,C 180,E1 -18364.433,E2 -18364.433} C_VEL
LIN {X 0,Y 274.784,Z 737.397,A -85,B 0,C 180,E1 -18366.289,E2 -18366.289} C_VEL
LIN {X 0,Y 275.431,Z 734.718,A -85,B 0,C 180,E1 -18367.378,E2 -18367.378} C_VEL
LIN {X 0,Y 275.06,Z 730.467,A -85,B 0,C 180,E1 -18369.243,E2 -18369.243} C_VEL
LIN {X 0,Y 274.807,Z 725.785,A -85,B 0,C 180,E1 -18371.053,E2 -18371.053} C_VEL
LIN {X 0,Y 275.598,Z 722.282,A -85,B 0,C 180,E1 -18372.033,E2 -18372.033} C_VEL
LIN {X 0,Y 278.501,Z 713.83,A -85,B 0,C 180,E1 -18373.871,E2 -18373.871} C_VEL
LIN {X 0,Y 281.774,Z 703.046,A -85,B 0,C 180,E1 -18375.739,E2 -18375.739} C_VEL
LIN {X 0,Y 284.455,Z 692.367,A -85,B 0,C 180,E1 -18377.247,E2 -18377.247} C_VEL
LIN {X 0,Y 286.947,Z 680.826,A -85,B 0,C 180,E1 -18378.567,E2 -18378.567} C_VEL
LIN {X 0,Y 288.979,Z 668.273,A -85,B 0,C 180,E1 -18379.722,E2 -18379.722} C_VEL
LIN {X 0,Y 290.514,Z 654.536,A -85,B 0,C 180,E1 -18380.692,E2 -18380.692} C_VEL
LIN {X 0,Y 291.756,Z 636.545,A -85,B 0,C 180,E1 -18381.572,E2 -18381.572} C_VEL
LIN {X 0,Y 293.077,Z 619.352,A -85,B 0,C 180,E1 -18382.28,E2 -18382.28} C_VEL
LIN {X 0,Y 289.476,Z 612.29,A -85,B 0,C 180,E1 -18383.867,E2 -18383.867} C_VEL
LIN {X 0,Y 285.432,Z 605.372,A -85,B 0,C 180,E1 -18385.887,E2 -18385.887} C_VEL
LIN {X 0,Y 282.51,Z 600.917,A -85,B 0,C 180,E1 -18387.583,E2 -18387.583} C_VEL
LIN {X 0,Y 280.318,Z 597.431,A -85,B 0,C 180,E1 -18389.119,E2 -18389.119} C_VEL
LIN {X 0,Y 277.691,Z 594.277,A -85,B 0,C 180,E1 -18391.289,E2 -18391.289} C_VEL
LIN {X 0,Y 276.752,Z 592.257,A -85,B 0,C 180,E1 -18392.462,E2 -18392.462} C_VEL
LIN {X 0,Y 274.434,Z 590.327,A -85,B 0,C 180,E1 -18396.338,E2 -18396.338} C_VEL
LIN {X 0,Y 274.17,Z 590.009,A -85,B 0,C 180,E1 -18397.968,E2 -18397.968} C_VEL
LIN {X 0,Y 274.524,Z 590.523,A -85,B 0,C 180,E1 -18400.598,E2 -18400.598} C_VEL
LIN {X 0,Y 276.867,Z 592.507,A -85,B 0,C 180,E1 -18404.312,E2 -18404.312} C_VEL
LIN {X 0,Y 278.469,Z 595.716,A -85,B 0,C 180,E1 -18406.136,E2 -18406.136} C_VEL
LIN {X 0,Y 279.263,Z 596.823,A -85,B 0,C 180,E1 -18406.831,E2 -18406.831} C_VEL
LIN {X 0,Y 281.731,Z 607.859,A -85,B 0,C 180,E1 -18409.493,E2 -18409.493} C_VEL
LIN {X 0,Y 283.59,Z 616.817,A -85,B 0,C 180,E1 -18411.183,E2 -18411.183} C_VEL
LIN {X 0,Y 284.852,Z 634.589,A -85,B 0,C 180,E1 -18413.175,E2 -18413.175} C_VEL
LIN {X 0,Y 285.849,Z 653.552,A -85,B 0,C 180,E1 -18414.935,E2 -18414.935} C_VEL
LIN {X 0,Y 286.121,Z 664.453,A -85,B 0,C 180,E1 -18415.793,E2 -18415.793} C_VEL
LIN {X 0,Y 285.984,Z 693.744,A -85,B 0,C 180,E1 -18417.684,E2 -18417.684} C_VEL
LIN {X 0,Y 283.924,Z 710.758,A -85,B 0,C 180,E1 -18418.454,E2 -18418.454} C_VEL
LIN {X 0,Y 281.037,Z 726.167,A -85,B 0,C 180,E1 -18419.369,E2 -18419.369} C_VEL
LIN {X 0,Y 277.88,Z 739.616,A -85,B 0,C 180,E1 -18420.451,E2 -18420.451} C_VEL
LIN {X 0,Y 274.059,Z 753.528,A -85,B 0,C 180,E1 -18421.888,E2 -18421.888} C_VEL
LIN {X 0,Y 270.306,Z 766.019,A -85,B 0,C 180,E1 -18423.562,E2 -18423.562} C_VEL
LIN {X 0,Y 266.566,Z 777.401,A -85,B 0,C 180,E1 -18425.466,E2 -18425.466} C_VEL
LIN {X 0,Y 263.163,Z 787.682,A -85,B 0,C 180,E1 -18427.633,E2 -18427.633} C_VEL
LIN {X 0,Y 260.387,Z 796.231,A -85,B 0,C 180,E1 -18429.872,E2 -18429.872} C_VEL
LIN {X 0,Y 257.882,Z 804.479,A -85,B 0,C 180,E1 -18432.557,E2 -18432.557} C_VEL
LIN {X 0,Y 256.413,Z 810.208,A -85,B 0,C 180,E1 -18434.908,E2 -18434.908} C_VEL
LIN {X 0,Y 255.409,Z 814.854,A -85,B 0,C 180,E1 -18437.284,E2 -18437.284} C_VEL
LIN {X 0,Y 255.007,Z 818.509,A -85,B 0,C 180,E1 -18439.681,E2 -18439.681} C_VEL
LIN {X 0,Y 255.116,Z 821.711,A -85,B 0,C 180,E1 -18442.633,E2 -18442.633} C_VEL
LIN {X 0,Y 255.656,Z 823.368,A -85,B 0,C 180,E1 -18445.27,E2 -18445.27} C_VEL
LIN {X 0,Y 255.994,Z 823.787,A -85,B 0,C 180,E1 -18446.853,E2 -18446.853} C_VEL
LIN {X 0,Y 256.674,Z 823.648,A -85,B 0,C 180,E1 -18449.216,E2 -18449.216} C_VEL
LIN {X 0,Y 256.799,Z 824.204,A -85,B 0,C 180,E1 -18450.001,E2 -18450.001} C_VEL
LIN {X 0,Y 256.254,Z 824.852,A -85,B 0,C 180,E1 -18451.573,E2 -18451.573} C_VEL
LIN {X 0,Y 255.824,Z 825.065,A -85,B 0,C 180,E1 -18453.151,E2 -18453.151} C_VEL
LIN {X 0,Y 255.511,Z 824.835,A -85,B 0,C 180,E1 -18454.734,E2 -18454.734} C_VEL
LIN {X 0,Y 254.923,Z 823.058,A -85,B 0,C 180,E1 -18457.924,E2 -18457.924} C_VEL
LIN {X 0,Y 254.943,Z 819.681,A -85,B 0,C 180,E1 -18461.127,E2 -18461.127} C_VEL
LIN {X 0,Y 255.949,Z 814.736,A -85,B 0,C 180,E1 -18464.309,E2 -18464.309} C_VEL
LIN {X 0,Y 257.548,Z 808.613,A -85,B 0,C 180,E1 -18467.235,E2 -18467.235} C_VEL
LIN {X 0,Y 260.42,Z 800.728,A -85,B 0,C 180,E1 -18470.127,E2 -18470.127} C_VEL
LIN {X 0,Y 263.924,Z 791.812,A -85,B 0,C 180,E1 -18472.714,E2 -18472.714} C_VEL
LIN {X 0,Y 267.493,Z 782.726,A -85,B 0,C 180,E1 -18474.859,E2 -18474.859} C_VEL
LIN {X 0,Y 271.668,Z 772.055,A -85,B 0,C 180,E1 -18476.919,E2 -18476.919} C_VEL
LIN {X 0,Y 276.195,Z 760.505,A -85,B 0,C 180,E1 -18478.705,E2 -18478.705} C_VEL
LIN {X 0,Y 281.119,Z 746.786,A -85,B 0,C 180,E1 -18480.415,E2 -18480.415} C_VEL
LIN {X 0,Y 286.038,Z 731.816,A -85,B 0,C 180,E1 -18481.889,E2 -18481.889} C_VEL
LIN {X 0,Y 290.566,Z 716.099,A -85,B 0,C 180,E1 -18483.075,E2 -18483.075} C_VEL
LIN {X 0,Y 294.339,Z 700.248,A -85,B 0,C 180,E1 -18484.03,E2 -18484.03} C_VEL
LIN {X 0,Y 295.811,Z 692.347,A -85,B 0,C 180,E1 -18484.455,E2 -18484.455} C_VEL
LIN {X 0,Y 298.33,Z 669.221,A -85,B 0,C 180,E1 -18485.824,E2 -18485.824} C_VEL
LIN {X 0,Y 299.339,Z 653.766,A -85,B 0,C 180,E1 -18487,E2 -18487} C_VEL
LIN {X 0,Y 299.974,Z 639.347,A -85,B 0,C 180,E1 -18488.4,E2 -18488.4} C_VEL
LIN {X 0,Y 300.534,Z 625.782,A -85,B 0,C 180,E1 -18490.014,E2 -18490.014} C_VEL
LIN {X 0,Y 300.739,Z 620.691,A -85,B 0,C 180,E1 -18490.742,E2 -18490.742} C_VEL
LIN {X 0,Y 299.151,Z 617.143,A -85,B 0,C 180,E1 -18493.46,E2 -18493.46} C_VEL
LIN {X 0,Y 299.033,Z 616.594,A -85,B 0,C 180,E1 -18493.956,E2 -18493.956} C_VEL
LIN {X 0,Y 298.902,Z 616.502,A -85,B 0,C 180,E1 -18497.009,E2 -18497.009} C_VEL
LIN {X 0,Y 299.326,Z 616.83,A -85,B 0,C 180,E1 -18498.099,E2 -18498.099} C_VEL
LIN {X 0,Y 300.759,Z 620.108,A -85,B 0,C 180,E1 -18500.456,E2 -18500.456} C_VEL
LIN {X 0,Y 301.439,Z 621.248,A -85,B 0,C 180,E1 -18501.158,E2 -18501.158} C_VEL
LIN {X 0,Y 303.321,Z 625.01,A -85,B 0,C 180,E1 -18502.781,E2 -18502.781} C_VEL
LIN {X 0,Y 305.184,Z 629.146,A -85,B 0,C 180,E1 -18504.109,E2 -18504.109} C_VEL
LIN {X 0,Y 303.21,Z 647.925,A -85,B 0,C 180,E1 -18505.064,E2 -18505.064} C_VEL
LIN {X 0,Y 301.166,Z 662.366,A -85,B 0,C 180,E1 -18506.04,E2 -18506.04} C_VEL
LIN {X 0,Y 298.539,Z 675.741,A -85,B 0,C 180,E1 -18507.217,E2 -18507.217} C_VEL
LIN {X 0,Y 295.296,Z 688.747,A -85,B 0,C 180,E1 -18508.625,E2 -18508.625} C_VEL
LIN {X 0,Y 292.099,Z 699.404,A -85,B 0,C 180,E1 -18510.048,E2 -18510.048} C_VEL
LIN {X 0,Y 287.958,Z 711.161,A -85,B 0,C 180,E1 -18511.967,E2 -18511.967} C_VEL
LIN {X 0,Y 283.975,Z 720.983,A -85,B 0,C 180,E1 -18513.941,E2 -18513.941} C_VEL
LIN {X 0,Y 279.643,Z 730.428,A -85,B 0,C 180,E1 -18516.289,E2 -18516.289} C_VEL
LIN {X 0,Y 276.18,Z 737.107,A -85,B 0,C 180,E1 -18518.346,E2 -18518.346} C_VEL
LIN {X 0,Y 272.995,Z 742.66,A -85,B 0,C 180,E1 -18520.447,E2 -18520.447} C_VEL
LIN {X 0,Y 269.161,Z 748.718,A -85,B 0,C 180,E1 -18523.308,E2 -18523.308} C_VEL
LIN {X 0,Y 265.856,Z 753.207,A -85,B 0,C 180,E1 -18526.236,E2 -18526.236} C_VEL
LIN {X 0,Y 263.019,Z 756.353,A -85,B 0,C 180,E1 -18529.219,E2 -18529.219} C_VEL
LIN {X 0,Y 260.925,Z 758.143,A -85,B 0,C 180,E1 -18532.26,E2 -18532.26} C_VEL
LIN {X 0,Y 259.129,Z 758.726,A -85,B 0,C 180,E1 -18535.332,E2 -18535.332} C_VEL
LIN {X 0,Y 257.874,Z 758.067,A -85,B 0,C 180,E1 -18538.438,E2 -18538.438} C_VEL
LIN {X 0,Y 257.083,Z 756.159,A -85,B 0,C 180,E1 -18541.566,E2 -18541.566} C_VEL
LIN {X 0,Y 256.515,Z 753,A -85,B 0,C 180,E1 -18544.714,E2 -18544.714} C_VEL
LIN {X 0,Y 256.647,Z 748.471,A -85,B 0,C 180,E1 -18547.869,E2 -18547.869} C_VEL
LIN {X 0,Y 256.909,Z 742.467,A -85,B 0,C 180,E1 -18551.039,E2 -18551.039} C_VEL
LIN {X 0,Y 257.381,Z 735.844,A -85,B 0,C 180,E1 -18553.822,E2 -18553.822} C_VEL
LIN {X 0,Y 258.291,Z 727.746,A -85,B 0,C 180,E1 -18556.6,E2 -18556.6} C_VEL
LIN {X 0,Y 259.396,Z 717.878,A -85,B 0,C 180,E1 -18559.383,E2 -18559.383} C_VEL
LIN {X 0,Y 260.629,Z 707.73,A -85,B 0,C 180,E1 -18561.763,E2 -18561.763} C_VEL
LIN {X 0,Y 262.138,Z 695.534,A -85,B 0,C 180,E1 -18564.138,E2 -18564.138} C_VEL
LIN {X 0,Y 263.533,Z 683.364,A -85,B 0,C 180,E1 -18566.105,E2 -18566.105} C_VEL
LIN {X 0,Y 264.956,Z 670.146,A -85,B 0,C 180,E1 -18567.872,E2 -18567.872} C_VEL
LIN {X 0,Y 266.233,Z 656.016,A -85,B 0,C 180,E1 -18569.408,E2 -18569.408} C_VEL
LIN {X 0,Y 267.258,Z 641.783,A -85,B 0,C 180,E1 -18570.63,E2 -18570.63} C_VEL
LIN {X 0,Y 268.13,Z 626.588,A -85,B 0,C 180,E1 -18571.615,E2 -18571.615} C_VEL
LIN {X 0,Y 268.672,Z 609.26,A -85,B 0,C 180,E1 -18572.409,E2 -18572.409} C_VEL
LIN {X 0,Y 268.636,Z 603.775,A -85,B 0,C 180,E1 -18572.638,E2 -18572.638} C_VEL
LIN {X 0,Y 256.123,Z 568.578,A -85,B 0,C 180,E1 -18575.004,E2 -18575.004} C_VEL
LIN {X 0,Y 256.123,Z 568.578,A -85,B 0,C 180,E1 -18577.272,E2 -18577.272} C_VEL
LIN {X 0,Y 256.072,Z 568.588,A -85,B 0,C 180,E1 -18582.18,E2 -18582.18} C_VEL
LIN {X 0,Y 256.064,Z 568.587,A -85,B 0,C 180,E1 -18586.672,E2 -18586.672} C_VEL
LIN {X 0,Y 256.091,Z 568.584,A -85,B 0,C 180,E1 -18590.86,E2 -18590.86} C_VEL
LIN {X 0,Y 256.121,Z 568.58,A -85,B 0,C 180,E1 -18594.812,E2 -18594.812} C_VEL
LIN {X 0,Y 256.092,Z 568.585,A -85,B 0,C 180,E1 -18598.571,E2 -18598.571} C_VEL
LIN {X 0,Y 256.137,Z 568.578,A -85,B 0,C 180,E1 -18602.195,E2 -18602.195} C_VEL
LIN {X 0,Y 256.166,Z 568.571,A -85,B 0,C 180,E1 -18605.698,E2 -18605.698} C_VEL
LIN {X 0,Y 256.166,Z 568.575,A -85,B 0,C 180,E1 -18609.104,E2 -18609.104} C_VEL
LIN {X 0,Y 256.299,Z 568.556,A -85,B 0,C 180,E1 -18614.084,E2 -18614.084} C_VEL
LIN {X 0,Y 256.308,Z 568.56,A -85,B 0,C 180,E1 -18618.933,E2 -18618.933} C_VEL
LIN {X 0,Y 256.539,Z 568.526,A -85,B 0,C 180,E1 -18622.126,E2 -18622.126} C_VEL
LIN {X 0,Y 256.713,Z 568.506,A -85,B 0,C 180,E1 -18628.43,E2 -18628.43} C_VEL
LIN {X 0,Y 256.713,Z 568.505,A -85,B 0,C 180,E1 -18631.568,E2 -18631.568} C_VEL
LIN {X 0,Y 256.537,Z 568.528,A -85,B 0,C 180,E1 -18637.872,E2 -18637.872} C_VEL
LIN {X 0,Y 256.307,Z 568.557,A -85,B 0,C 180,E1 -18641.065,E2 -18641.065} C_VEL
LIN {X 0,Y 256.296,Z 568.558,A -85,B 0,C 180,E1 -18645.914,E2 -18645.914} C_VEL
LIN {X 0,Y 256.214,Z 568.566,A -85,B 0,C 180,E1 -18650.89,E2 -18650.89} C_VEL
LIN {X 0,Y 256.184,Z 568.572,A -85,B 0,C 180,E1 -18655.138,E2 -18655.138} C_VEL
LIN {X 0,Y 256.107,Z 568.583,A -85,B 0,C 180,E1 -18659.599,E2 -18659.599} C_VEL
LIN {X 0,Y 256.081,Z 568.585,A -85,B 0,C 180,E1 -18663.29,E2 -18663.29} C_VEL
LIN {X 0,Y 256.136,Z 568.578,A -85,B 0,C 180,E1 -18667.278,E2 -18667.278} C_VEL
LIN {X 0,Y 256.084,Z 568.584,A -85,B 0,C 180,E1 -18671.196,E2 -18671.196} C_VEL
LIN {X 0,Y 256.108,Z 568.582,A -85,B 0,C 180,E1 -18674.482,E2 -18674.482} C_VEL
LIN {X 0,Y 256.182,Z 568.573,A -85,B 0,C 180,E1 -18677.447,E2 -18677.447} C_VEL
LIN {X 0,Y 267.744,Z 600.325,A -85,B 0,C 180,E1 -18679.498,E2 -18679.498} C_VEL
LIN {X 0,Y 266.931,Z 633.918,A -85,B 0,C 180,E1 -18680.778,E2 -18680.778} C_VEL
LIN {X 0,Y 266.305,Z 647.552,A -85,B 0,C 180,E1 -18681.551,E2 -18681.551} C_VEL
LIN {X 0,Y 265.495,Z 660.735,A -85,B 0,C 180,E1 -18682.572,E2 -18682.572} C_VEL
LIN {X 0,Y 264.357,Z 674.55,A -85,B 0,C 180,E1 -18683.972,E2 -18683.972} C_VEL
LIN {X 0,Y 262.989,Z 687.576,A -85,B 0,C 180,E1 -18685.631,E2 -18685.631} C_VEL
LIN {X 0,Y 261.673,Z 699.452,A -85,B 0,C 180,E1 -18687.51,E2 -18687.51} C_VEL
LIN {X 0,Y 260.342,Z 710.241,A -85,B 0,C 180,E1 -18689.6,E2 -18689.6} C_VEL
LIN {X 0,Y 259.087,Z 720.82,A -85,B 0,C 180,E1 -18692.101,E2 -18692.101} C_VEL
LIN {X 0,Y 258.042,Z 729.414,A -85,B 0,C 180,E1 -18694.599,E2 -18694.599} C_VEL
LIN {X 0,Y 257.164,Z 737.43,A -85,B 0,C 180,E1 -18697.506,E2 -18697.506} C_VEL
LIN {X 0,Y 256.667,Z 742.91,A -85,B 0,C 180,E1 -18699.985,E2 -18699.985} C_VEL
LIN {X 0,Y 256.377,Z 747.251,A -85,B 0,C 180,E1 -18702.451,E2 -18702.451} C_VEL
LIN {X 0,Y 256.412,Z 751.483,A -85,B 0,C 180,E1 -18705.72,E2 -18705.72} C_VEL
LIN {X 0,Y 256.592,Z 752.987,A -85,B 0,C 180,E1 -18707.343,E2 -18707.343} C_VEL
LIN {X 0,Y 257.245,Z 754.795,A -85,B 0,C 180,E1 -18710.566,E2 -18710.566} C_VEL
LIN {X 0,Y 258.336,Z 755.139,A -85,B 0,C 180,E1 -18713.753,E2 -18713.753} C_VEL
LIN {X 0,Y 259.883,Z 754.024,A -85,B 0,C 180,E1 -18716.9,E2 -18716.9} C_VEL
LIN {X 0,Y 261.949,Z 751.379,A -85,B 0,C 180,E1 -18720.001,E2 -18720.001} C_VEL
LIN {X 0,Y 264.55,Z 747.184,A -85,B 0,C 180,E1 -18723.046,E2 -18723.046} C_VEL
LIN {X 0,Y 266.764,Z 742.934,A -85,B 0,C 180,E1 -18725.291,E2 -18725.291} C_VEL
LIN {X 0,Y 269.408,Z 737.469,A -85,B 0,C 180,E1 -18727.572,E2 -18727.572} C_VEL
LIN {X 0,Y 272.697,Z 729.979,A -85,B 0,C 180,E1 -18730.019,E2 -18730.019} C_VEL
LIN {X 0,Y 275.598,Z 722.282,A -85,B 0,C 180,E1 -18732.033,E2 -18732.033} C_VEL
LIN {X 0,Y 276.422,Z 718.66,A -85,B 0,C 180,E1 -18732.991,E2 -18732.991} C_VEL
LIN {X 0,Y 276.404,Z 712.917,A -85,B 0,C 180,E1 -18734.67,E2 -18734.67} C_VEL
LIN {X 0,Y 276.501,Z 706.734,A -85,B 0,C 180,E1 -18736.261,E2 -18736.261} C_VEL
LIN {X 0,Y 277.39,Z 702.417,A -85,B 0,C 180,E1 -18737.066,E2 -18737.066} C_VEL
LIN {X 0,Y 280.089,Z 692.304,A -85,B 0,C 180,E1 -18738.469,E2 -18738.469} C_VEL
LIN {X 0,Y 282.672,Z 680.38,A -85,B 0,C 180,E1 -18739.802,E2 -18739.802} C_VEL
LIN {X 0,Y 284.971,Z 666.353,A -85,B 0,C 180,E1 -18741.048,E2 -18741.048} C_VEL
LIN {X 0,Y 286.51,Z 652.948,A -85,B 0,C 180,E1 -18741.938,E2 -18741.938} C_VEL
LIN {X 0,Y 287.965,Z 633.032,A -85,B 0,C 180,E1 -18742.883,E2 -18742.883} C_VEL
LIN {X 0,Y 288.815,Z 622.728,A -85,B 0,C 180,E1 -18743.331,E2 -18743.331} C_VEL
LIN {X 0,Y 285.868,Z 616.971,A -85,B 0,C 180,E1 -18744.748,E2 -18744.748} C_VEL
LIN {X 0,Y 282.264,Z 610.676,A -85,B 0,C 180,E1 -18746.727,E2 -18746.727} C_VEL
LIN {X 0,Y 280.059,Z 607.096,A -85,B 0,C 180,E1 -18748.132,E2 -18748.132} C_VEL
LIN {X 0,Y 278.04,Z 603.697,A -85,B 0,C 180,E1 -18749.677,E2 -18749.677} C_VEL
LIN {X 0,Y 275.758,Z 600.758,A -85,B 0,C 180,E1 -18751.734,E2 -18751.734} C_VEL
LIN {X 0,Y 275.098,Z 599.115,A -85,B 0,C 180,E1 -18752.682,E2 -18752.682} C_VEL
LIN {X 0,Y 272.921,Z 597.199,A -85,B 0,C 180,E1 -18756.572,E2 -18756.572} C_VEL
LIN {X 0,Y 272.758,Z 597.084,A -85,B 0,C 180,E1 -18759.378,E2 -18759.378} C_VEL
LIN {X 0,Y 274.333,Z 598.708,A -85,B 0,C 180,E1 -18763.09,E2 -18763.09} C_VEL
LIN {X 0,Y 275.103,Z 599.389,A -85,B 0,C 180,E1 -18764.038,E2 -18764.038} C_VEL
LIN {X 0,Y 276.681,Z 602.504,A -85,B 0,C 180,E1 -18765.914,E2 -18765.914} C_VEL
LIN {X 0,Y 276.987,Z 603.215,A -85,B 0,C 180,E1 -18766.25,E2 -18766.25} C_VEL
LIN {X 0,Y 278.818,Z 612.7,A -85,B 0,C 180,E1 -18768.606,E2 -18768.606} C_VEL
LIN {X 0,Y 280.301,Z 621.075,A -85,B 0,C 180,E1 -18770.226,E2 -18770.226} C_VEL
LIN {X 0,Y 281.161,Z 639.088,A -85,B 0,C 180,E1 -18772.261,E2 -18772.261} C_VEL
LIN {X 0,Y 281.822,Z 656.823,A -85,B 0,C 180,E1 -18773.947,E2 -18773.947} C_VEL
LIN {X 0,Y 281.892,Z 667.546,A -85,B 0,C 180,E1 -18774.785,E2 -18774.785} C_VEL
LIN {X 0,Y 281.367,Z 695.272,A -85,B 0,C 180,E1 -18776.616,E2 -18776.616} C_VEL
LIN {X 0,Y 279.125,Z 711.55,A -85,B 0,C 180,E1 -18777.407,E2 -18777.407} C_VEL
LIN {X 0,Y 276.043,Z 726.234,A -85,B 0,C 180,E1 -18778.326,E2 -18778.326} C_VEL
LIN {X 0,Y 272.29,Z 740.975,A -85,B 0,C 180,E1 -18779.568,E2 -18779.568} C_VEL
LIN {X 0,Y 268.344,Z 754.208,A -85,B 0,C 180,E1 -18781.02,E2 -18781.02} C_VEL
LIN {X 0,Y 264.42,Z 766.265,A -85,B 0,C 180,E1 -18782.712,E2 -18782.712} C_VEL
